C05446=1014.097,308.316,353.938,169.733,52.430,160.170
C05447=1014.104,308.600,353.902,169.740,52.424,160.169
C05448=1014.111,308.846,353.870,169.746,52.418,160.169
C05449=1014.117,309.094,353.839,169.753,52.412,160.169
C05450=1014.123,309.343,353.807,169.760,52.406,160.169
C05451=1014.128,309.590,353.774,169.766,52.401,160.169
C05452=1014.134,309.838,353.742,169.772,52.395,160.169
C05453=1014.141,310.086,353.709,169.779,52.389,160.169
C05454=1014.147,310.333,353.676,169.785,52.384,160.169
C05455=1014.153,310.581,353.644,169.792,52.379,160.169
C05456=1014.158,310.829,353.611,169.798,52.373,160.169
C05457=1014.164,311.077,353.579,169.804,52.367,160.169
C05458=1014.170,311.324,353.547,169.811,52.362,160.169
C05459=1014.176,311.572,353.514,169.817,52.356,160.169
C05460=1014.182,311.820,353.482,169.824,52.350,160.169
C05461=1014.189,312.068,353.449,169.831,52.345,160.169
C05462=1014.194,312.315,353.416,169.837,52.339,160.169
C05463=1014.200,312.563,353.384,169.843,52.333,160.169
C05464=1014.206,312.811,353.351,169.850,52.328,160.169
C05465=1014.212,313.058,353.319,169.856,52.323,160.169
C05466=1014.218,313.306,353.286,169.863,52.317,160.169
C05467=1014.224,313.554,353.254,169.869,52.311,160.169
C05468=1014.230,313.802,353.220,169.876,52.306,160.169
C05469=1014.236,314.050,353.188,169.883,52.300,160.169
C05470=1014.243,314.297,353.155,169.889,52.295,160.169
C05471=1014.249,314.545,353.122,169.896,52.290,160.169
C05472=1014.255,314.792,353.089,169.902,52.284,160.169
C05473=1014.261,315.040,353.056,169.909,52.278,160.169
C05474=1014.267,315.289,353.024,169.915,52.273,160.169
C05475=1014.273,315.536,352.991,169.922,52.268,160.169
C05476=1014.279,315.784,352.959,169.928,52.263,160.169
C05477=1014.286,316.031,352.926,169.936,52.257,160.169
C05478=1014.292,316.279,352.893,169.942,52.252,160.169
C05479=1014.297,316.527,352.860,169.949,52.246,160.169
C05480=1014.304,316.775,352.827,169.955,52.241,160.169
C05481=1014.311,317.023,352.794,169.962,52.236,160.169
C05482=1014.317,317.270,352.761,169.968,52.231,160.169
C05483=1014.323,317.518,352.728,169.975,52.225,160.169
C05484=1014.329,317.766,352.695,169.982,52.220,160.169
C05485=1014.335,318.013,352.662,169.989,52.214,160.169
C05486=1014.342,318.260,352.629,169.995,52.209,160.169
C05487=1014.348,318.509,352.596,170.002,52.203,160.169
C05488=1014.355,318.756,352.563,170.008,52.198,160.169
C05489=1014.360,319.004,352.530,170.015,52.193,160.169
C05490=1014.367,319.252,352.497,170.022,52.187,160.169
C05491=1014.374,319.499,352.463,170.029,52.182,160.169
C05492=1014.380,319.747,352.430,170.036,52.177,160.170
C05493=1014.386,319.995,352.398,170.042,52.172,160.169
C05494=1014.392,320.243,352.364,170.049,52.167,160.170
C05495=1014.399,320.490,352.331,170.056,52.162,160.170
C05496=1014.405,320.738,352.298,170.063,52.156,160.170
C05497=1014.412,320.985,352.265,170.070,52.151,160.170
C05498=1014.419,321.233,352.231,170.076,52.146,160.170
C05499=1014.425,321.481,352.198,170.083,52.141,160.170
C05500=1014.431,321.729,352.165,170.090,52.136,160.170
C05501=1014.438,321.976,352.131,170.096,52.131,160.170
C05502=1014.444,322.224,352.099,170.104,52.125,160.170
C05503=1014.452,322.472,352.065,170.110,52.120,160.170
C05504=1014.458,322.761,352.026,170.118,52.114,160.171
C05505=1014.466,323.050,351.987,170.126,52.108,160.171
C05506=1014.474,323.339,351.948,170.135,52.102,160.171
C05507=1014.481,323.628,351.909,170.143,52.096,160.171
C05508=1014.488,323.876,351.876,170.149,52.091,160.171
C05509=1014.495,324.123,351.842,170.156,52.086,160.171
C05510=1014.501,324.372,351.809,170.164,52.081,160.171
C05511=1014.507,324.619,351.775,170.170,52.076,160.172
C05512=1014.515,324.867,351.741,170.177,52.071,160.172
C05513=1014.521,325.114,351.709,170.184,52.066,160.172
C05514=1014.528,325.362,351.675,170.192,52.061,160.172
C05515=1014.535,325.609,351.641,170.198,52.056,160.172
C05516=1014.541,325.857,351.608,170.205,52.051,160.172
C05517=1014.547,326.104,351.574,170.212,52.046,160.172
C05518=1014.554,326.352,351.540,170.219,52.042,160.173
C05519=1014.560,326.600,351.505,170.226,52.037,160.173
C05520=1014.567,326.847,351.472,170.233,52.031,160.173
C05521=1014.573,327.095,351.437,170.240,52.026,160.173
C05522=1014.579,327.343,351.403,170.247,52.022,160.174
C05523=1014.586,327.590,351.369,170.254,52.017,160.174
C05524=1014.593,327.838,351.335,170.261,52.012,160.174
C05525=1014.599,328.085,351.301,170.268,52.008,160.174
C05526=1014.606,328.333,351.267,170.275,52.003,160.174
C05527=1014.612,328.580,351.232,170.283,51.998,160.175
C05528=1014.619,328.828,351.198,170.290,51.993,160.175
C05529=1014.626,329.075,351.164,170.296,51.988,160.175
C05530=1014.632,329.323,351.130,170.303,51.984,160.175
C05531=1014.638,329.571,351.096,170.310,51.979,160.175
C05532=1014.645,329.818,351.062,170.318,51.974,160.176
C05533=1014.652,330.066,351.027,170.325,51.969,160.176
C05534=1014.658,330.313,350.993,170.332,51.965,160.176
C05535=1014.665,330.561,350.959,170.339,51.960,160.176
C05536=1014.672,330.809,350.924,170.346,51.956,160.177
C05537=1014.678,331.056,350.889,170.353,51.951,160.177
C05538=1014.686,331.304,350.855,170.361,51.946,160.177
C05539=1014.691,331.551,350.821,170.368,51.942,160.178
C05540=1014.698,331.798,350.786,170.375,51.937,160.178
C05541=1014.705,332.046,350.752,170.382,51.933,160.178
C05542=1014.712,332.293,350.717,170.389,51.928,160.178
C05543=1014.719,332.541,350.683,170.397,51.923,160.178
C05544=1014.725,332.789,350.648,170.404,51.919,160.179
C05545=1014.731,333.036,350.614,170.411,51.914,160.179
C05546=1014.738,333.283,350.579,170.418,51.910,160.179
C05547=1014.745,333.531,350.543,170.425,51.905,160.180
C05548=1014.751,333.779,350.509,170.433,51.901,160.180
C05549=1014.759,334.026,350.474,170.440,51.896,160.180
C05550=1014.766,334.273,350.439,170.448,51.892,160.181
C05551=1014.772,334.521,350.405,170.455,51.888,160.181
C05552=1014.779,334.769,350.370,170.462,51.883,160.181
C05553=1014.786,335.016,350.335,170.470,51.878,160.182
C05554=1014.792,335.263,350.300,170.477,51.874,160.182
C05555=1014.799,335.511,350.265,170.484,51.870,160.182
C05556=1014.806,335.759,350.230,170.491,51.865,160.182
C05557=1014.812,336.006,350.195,170.498,51.861,160.183
C05558=1014.819,336.253,350.160,170.506,51.856,160.183
C05559=1014.826,336.501,350.125,170.513,51.852,160.184
C05560=1014.833,336.748,350.089,170.521,51.848,160.184
C05561=1014.839,336.995,350.054,170.528,51.843,160.184
C05562=1014.846,337.243,350.020,170.535,51.839,160.185
C05563=1014.853,337.491,349.985,170.543,51.834,160.185
C05564=1014.861,337.776,349.944,170.551,51.830,160.185
C05565=1014.869,338.060,349.903,170.560,51.825,160.186
C05566=1014.877,338.345,349.864,170.569,51.820,160.186
C05567=1014.885,338.630,349.823,170.578,51.815,160.187
C05568=1014.892,338.878,349.788,170.585,51.811,160.187
C05569=1014.899,339.125,349.752,170.592,51.807,160.187
C05570=1014.905,339.372,349.716,170.600,51.803,160.188
C05571=1014.912,339.619,349.681,170.608,51.798,160.188
C05572=1014.919,339.867,349.645,170.615,51.794,160.189
C05573=1014.926,340.114,349.610,170.623,51.790,160.189
C05574=1014.933,340.362,349.574,170.630,51.786,160.190
C05575=1014.940,340.609,349.539,170.638,51.781,160.190
C05576=1014.946,340.856,349.503,170.645,51.778,160.191
C05577=1014.954,341.104,349.467,170.653,51.773,160.191
C05578=1014.960,341.351,349.432,170.660,51.770,160.191
C05579=1014.967,341.598,349.396,170.668,51.765,160.192
C05580=1014.975,341.846,349.361,170.675,51.761,160.192
C05581=1014.981,342.093,349.324,170.683,51.757,160.193
C05582=1014.988,342.341,349.289,170.690,51.753,160.193
C05583=1014.996,342.588,349.253,170.699,51.749,160.194
C05584=1015.002,342.835,349.218,170.706,51.745,160.194
C05585=1015.009,343.083,349.181,170.714,51.741,160.194
C05586=1015.016,343.330,349.145,170.721,51.737,160.195
C05587=1015.023,343.577,349.110,170.729,51.733,160.195
C05588=1015.030,343.825,349.073,170.737,51.729,160.196
C05589=1015.037,344.072,349.037,170.744,51.726,160.197
C05590=1015.044,344.319,349.002,170.753,51.721,160.197
C05591=1015.052,344.567,348.966,170.760,51.717,160.197
C05592=1015.058,344.814,348.930,170.768,51.714,160.198
C05593=1015.066,345.061,348.893,170.776,51.709,160.198
C05594=1015.072,345.309,348.858,170.783,51.705,160.199
C05595=1015.080,345.556,348.822,170.791,51.702,160.199
C05596=1015.086,345.803,348.786,170.799,51.698,160.200
C05597=1015.094,346.050,348.749,170.807,51.694,160.201
C05598=1015.101,346.297,348.714,170.814,51.690,160.201
C05599=1015.108,346.545,348.677,170.822,51.686,160.201
C05600=1015.116,346.792,348.641,170.830,51.682,160.202
C05601=1015.122,347.039,348.604,170.838,51.679,160.203
C05602=1015.130,347.287,348.568,170.846,51.675,160.203
C05603=1015.137,347.534,348.532,170.854,51.671,160.204
C05604=1015.144,347.781,348.495,170.862,51.667,160.204
C05605=1015.151,348.028,348.459,170.869,51.664,160.205
C05606=1015.158,348.276,348.423,170.878,51.660,160.206
C05607=1015.165,348.523,348.385,170.886,51.656,160.206
C05608=1015.172,348.770,348.349,170.893,51.652,160.207
C05609=1015.179,349.018,348.312,170.902,51.649,160.207
C05610=1015.187,349.265,348.276,170.909,51.645,160.208
C05611=1015.193,349.511,348.239,170.917,51.641,160.208
C05612=1015.201,349.759,348.203,170.926,51.638,160.209
C05613=1015.208,350.007,348.166,170.933,51.634,160.210
C05614=1015.216,350.253,348.129,170.942,51.630,160.210
C05615=1015.222,350.500,348.093,170.950,51.627,160.211
C05616=1015.230,350.747,348.056,170.957,51.623,160.211
C05617=1015.237,350.995,348.019,170.966,51.620,160.212
C05618=1015.245,351.243,347.983,170.974,51.616,160.213
C05619=1015.252,351.490,347.945,170.981,51.612,160.213
C05620=1015.259,351.736,347.909,170.990,51.609,160.214
C05621=1015.266,351.984,347.872,170.998,51.605,160.215
C05622=1015.274,352.231,347.834,171.006,51.601,160.215
C05623=1015.281,352.478,347.798,171.014,51.598,160.216
C05624=1015.290,352.760,347.756,171.024,51.594,160.217
C05625=1015.299,353.042,347.713,171.033,51.590,160.217
C05626=1015.307,353.325,347.671,171.043,51.586,160.218
C05627=1015.315,353.607,347.629,171.052,51.582,160.219
C05628=1015.322,353.854,347.592,171.060,51.579,160.220
C05629=1015.330,354.100,347.555,171.068,51.575,160.220
C05630=1015.337,354.348,347.517,171.077,51.572,160.221
C05631=1015.344,354.595,347.480,171.084,51.568,160.222
C05632=1015.352,354.842,347.442,171.093,51.565,160.222
C05633=1015.360,355.089,347.405,171.101,51.561,160.223
C05634=1015.367,355.336,347.368,171.110,51.558,160.224
C05635=1015.374,355.584,347.331,171.118,51.555,160.224
C05636=1015.382,355.831,347.293,171.126,51.551,160.225
C05637=1015.390,356.078,347.255,171.134,51.548,160.226
C05638=1015.397,356.325,347.218,171.143,51.545,160.227
C05639=1015.405,356.572,347.180,171.151,51.542,160.227
C05640=1015.412,356.819,347.143,171.160,51.538,160.228
C05641=1015.420,357.066,347.106,171.168,51.535,160.229
C05642=1015.427,357.313,347.068,171.177,51.532,160.230
C05643=1015.434,357.560,347.031,171.185,51.529,160.230
C05644=1015.442,357.807,346.992,171.194,51.525,160.231
C05645=1015.450,358.054,346.955,171.202,51.522,160.232
C05646=1015.458,358.301,346.918,171.211,51.519,160.233
C05647=1015.465,358.548,346.880,171.219,51.516,160.233
C05648=1015.472,358.795,346.842,171.227,51.512,160.234
C05649=1015.480,359.043,346.804,171.236,51.510,160.235
C05650=1015.488,359.289,346.766,171.245,51.506,160.236
C05651=1015.495,359.536,346.728,171.253,51.503,160.237
C05652=1015.503,359.783,346.690,171.262,51.500,160.237
C05653=1015.510,360.030,346.652,171.270,51.497,160.238
C05654=1015.518,360.277,346.614,171.279,51.494,160.239
C05655=1015.525,360.524,346.576,171.287,51.491,160.240
C05656=1015.533,360.771,346.538,171.296,51.487,160.241
C05657=1015.541,361.018,346.499,171.304,51.485,160.242
C05658=1015.548,361.265,346.461,171.313,51.482,160.242
C05659=1015.556,361.512,346.424,171.322,51.478,160.243
C05660=1015.563,361.759,346.384,171.330,51.475,160.244
C05661=1015.571,362.006,346.346,171.339,51.472,160.245
C05662=1015.579,362.253,346.308,171.347,51.469,160.246
C05663=1015.586,362.500,346.270,171.356,51.466,160.247
C05664=1015.594,362.747,346.232,171.366,51.463,160.248
C05665=1015.602,362.994,346.193,171.374,51.460,160.248
C05666=1015.609,363.240,346.155,171.383,51.457,160.249
C05667=1015.617,363.488,346.116,171.391,51.455,160.250
C05668=1015.625,363.734,346.078,171.400,51.451,160.251
C05669=1015.633,363.981,346.040,171.410,51.449,160.252
C05670=1015.641,364.228,346.001,171.418,51.446,160.253
C05671=1015.649,364.475,345.963,171.427,51.443,160.254
C05672=1015.657,364.722,345.924,171.436,51.440,160.255
C05673=1015.665,364.969,345.886,171.444,51.437,160.256
C05674=1015.673,365.216,345.847,171.453,51.434,160.256
C05675=1015.680,365.463,345.809,171.463,51.431,160.257
C05676=1015.689,365.709,345.770,171.471,51.429,160.258
C05677=1015.696,365.957,345.730,171.480,51.425,160.259
C05678=1015.704,366.203,345.692,171.489,51.423,160.260
C05679=1015.712,366.450,345.654,171.499,51.420,160.261
C05680=1015.720,366.697,345.614,171.507,51.417,160.262
C05681=1015.728,366.944,345.576,171.516,51.414,160.263
C05682=1015.736,367.191,345.537,171.526,51.412,160.264
C05683=1015.744,367.437,345.498,171.534,51.409,160.265
C05684=1015.753,367.727,345.452,171.545,51.406,160.266
C05685=1015.763,368.017,345.406,171.556,51.403,160.267
C05686=1015.772,368.307,345.361,171.566,51.400,160.268
C05687=1015.781,368.596,345.315,171.577,51.396,160.270
C05688=1015.789,368.843,345.275,171.586,51.394,160.271
C05689=1015.797,369.090,345.236,171.595,51.391,160.272
C05690=1015.806,369.336,345.196,171.605,51.388,160.273
C05691=1015.813,369.584,345.157,171.613,51.386,160.274
C05692=1015.821,369.831,345.118,171.623,51.383,160.275
C05693=1015.829,370.077,345.078,171.632,51.380,160.276
C05694=1015.837,370.323,345.039,171.642,51.378,160.277
C05695=1015.845,370.570,345.000,171.651,51.376,160.278
C05696=1015.853,370.817,344.960,171.660,51.373,160.279
C05697=1015.861,371.064,344.921,171.669,51.371,160.280
C05698=1015.869,371.311,344.881,171.678,51.368,160.281
C05699=1015.878,371.558,344.842,171.688,51.366,160.282
C05700=1015.886,371.804,344.803,171.698,51.363,160.283
C05701=1015.894,372.051,344.763,171.707,51.360,160.284
C05702=1015.902,372.298,344.723,171.715,51.358,160.285
C05703=1015.911,372.544,344.683,171.725,51.356,160.287
C05704=1015.919,372.791,344.643,171.735,51.353,160.288
C05705=1015.927,373.037,344.604,171.744,51.351,160.289
C05706=1015.935,373.284,344.564,171.754,51.348,160.290
C05707=1015.943,373.531,344.525,171.763,51.346,160.291
C05708=1015.952,373.778,344.485,171.773,51.343,160.292
C05709=1015.960,374.024,344.444,171.782,51.341,160.293
C05710=1015.969,374.271,344.405,171.792,51.339,160.294
C05711=1015.977,374.518,344.365,171.801,51.336,160.295
C05712=1015.985,374.764,344.325,171.811,51.334,160.297
C05713=1015.994,375.011,344.285,171.821,51.332,160.298
C05714=1016.002,375.258,344.246,171.830,51.329,160.299
C05715=1016.011,375.504,344.205,171.840,51.327,160.300
C05716=1016.019,375.751,344.166,171.850,51.325,160.302
C05717=1016.027,375.998,344.125,171.859,51.322,160.303
C05718=1016.036,376.244,344.085,171.868,51.320,160.304
C05719=1016.044,376.491,344.045,171.878,51.318,160.305
C05720=1016.052,376.737,344.004,171.888,51.316,160.306
C05721=1016.060,376.984,343.963,171.898,51.314,160.307
C05722=1016.069,377.230,343.923,171.907,51.311,160.308
C05723=1016.077,377.476,343.882,171.917,51.309,160.310
C05724=1016.085,377.724,343.842,171.927,51.307,160.311
C05725=1016.093,377.970,343.801,171.937,51.304,160.312
C05726=1016.102,378.216,343.761,171.947,51.302,160.314
C05727=1016.111,378.463,343.720,171.957,51.300,160.315
C05728=1016.119,378.709,343.680,171.967,51.298,160.316
C05729=1016.128,378.956,343.639,171.977,51.296,160.317
C05730=1016.136,379.202,343.599,171.986,51.294,160.319
C05731=1016.145,379.449,343.558,171.997,51.292,160.320
C05732=1016.153,379.696,343.517,172.006,51.290,160.321
C05733=1016.163,379.942,343.476,172.016,51.288,160.323
C05734=1016.171,380.188,343.435,172.026,51.286,160.324
C05735=1016.179,380.435,343.394,172.036,51.284,160.325
C05736=1016.187,380.681,343.354,172.047,51.282,160.327
C05737=1016.197,380.928,343.313,172.057,51.280,160.328
C05738=1016.206,381.174,343.272,172.067,51.278,160.329
C05739=1016.214,381.421,343.231,172.076,51.276,160.330
C05740=1016.222,381.668,343.190,172.087,51.274,160.332
C05741=1016.231,381.913,343.149,172.097,51.272,160.333
C05742=1016.240,382.160,343.108,172.108,51.270,160.335
C05743=1016.249,382.407,343.067,172.117,51.268,160.336
C05744=1016.260,382.719,343.015,172.130,51.265,160.338
C05745=1016.271,383.031,342.963,172.143,51.263,160.339
C05746=1016.282,383.343,342.910,172.156,51.261,160.341
C05747=1016.294,383.656,342.859,172.169,51.258,160.343
C05748=1016.303,383.903,342.817,172.179,51.256,160.344
C05749=1016.311,384.148,342.776,172.190,51.254,160.346
C05750=1016.321,384.395,342.735,172.201,51.253,160.347
C05751=1016.330,384.641,342.693,172.210,51.251,160.348
C05752=1016.338,384.888,342.652,172.222,51.249,160.350
C05753=1016.347,385.134,342.610,172.232,51.247,160.351
C05754=1016.356,385.381,342.568,172.242,51.246,160.353
C05755=1016.365,385.627,342.527,172.253,51.243,160.354
C05756=1016.374,385.873,342.485,172.263,51.242,160.356
C05757=1016.383,386.120,342.443,172.273,51.240,160.357
C05758=1016.392,386.366,342.401,172.284,51.238,160.359
C05759=1016.401,386.612,342.360,172.295,51.237,160.360
C05760=1016.409,386.858,342.318,172.305,51.235,160.362
C05761=1016.419,387.105,342.276,172.316,51.234,160.363
C05762=1016.428,387.351,342.235,172.326,51.232,160.365
C05763=1016.437,387.598,342.193,172.337,51.230,160.366
C05764=1016.446,387.844,342.150,172.348,51.229,160.368
C05765=1016.455,388.090,342.109,172.359,51.227,160.369
C05766=1016.464,388.336,342.066,172.369,51.226,160.371
C05767=1016.473,388.582,342.025,172.380,51.224,160.372
C05768=1016.482,388.828,341.983,172.391,51.222,160.374
C05769=1016.490,389.074,341.940,172.401,51.221,160.375
C05770=1016.499,389.321,341.898,172.413,51.220,160.377
C05771=1016.509,389.567,341.855,172.423,51.218,160.378
C05772=1016.519,389.813,341.813,172.434,51.216,160.380
C05773=1016.527,390.059,341.771,172.446,51.215,160.382
C05774=1016.537,390.305,341.729,172.456,51.213,160.383
C05775=1016.547,390.552,341.686,172.467,51.212,160.385
C05776=1016.555,390.798,341.644,172.478,51.210,160.386
C05777=1016.564,391.044,341.601,172.489,51.209,160.388
C05778=1016.574,391.290,341.558,172.499,51.208,160.390
C05779=1016.583,391.536,341.516,172.511,51.206,160.391
C05780=1016.592,391.783,341.474,172.522,51.204,160.393
C05781=1016.602,392.029,341.431,172.533,51.203,160.395
C05782=1016.610,392.275,341.388,172.544,51.202,160.396
C05783=1016.620,392.522,341.346,172.555,51.200,160.398
C05784=1016.630,392.767,341.302,172.566,51.199,160.400
C05785=1016.639,393.012,341.260,172.578,51.198,160.401
C05786=1016.648,393.259,341.217,172.589,51.197,160.403
C05787=1016.657,393.505,341.174,172.599,51.195,160.405
C05788=1016.667,393.751,341.131,172.611,51.194,160.406
C05789=1016.676,393.997,341.088,172.623,51.192,160.408
C05790=1016.686,394.243,341.045,172.633,51.192,160.410
C05791=1016.696,394.490,341.002,172.645,51.190,160.412
C05792=1016.704,394.736,340.959,172.656,51.189,160.413
C05793=1016.714,394.982,340.916,172.668,51.188,160.415
C05794=1016.724,395.227,340.873,172.680,51.186,160.417
C05795=1016.733,395.473,340.829,172.690,51.185,160.419
C05796=1016.743,395.720,340.786,172.702,51.184,160.420
C05797=1016.752,395.965,340.743,172.713,51.183,160.422
C05798=1016.761,396.212,340.700,172.725,51.182,160.424
C05799=1016.772,396.458,340.656,172.737,51.181,160.426
C05800=1016.782,396.703,340.613,172.749,51.179,160.428
C05801=1016.790,396.949,340.570,172.760,51.178,160.429
C05802=1016.800,397.195,340.526,172.771,51.178,160.431
C05803=1016.810,397.441,340.482,172.783,51.176,160.433
C05804=1016.824,397.787,340.421,172.799,51.175,160.436
C05805=1016.837,398.133,340.359,172.816,51.174,160.438
C05806=1016.851,398.479,340.298,172.832,51.172,160.441
C05807=1016.865,398.826,340.236,172.849,51.170,160.443
C05808=1016.874,399.071,340.193,172.861,51.170,160.445
C05809=1016.884,399.318,340.149,172.873,51.169,160.447
C05810=1016.894,399.563,340.105,172.884,51.168,160.449
C05811=1016.904,399.809,340.060,172.896,51.167,160.451
C05812=1016.914,400.055,340.017,172.909,51.166,160.453
C05813=1016.923,400.301,339.973,172.921,51.164,160.455
C05814=1016.934,400.547,339.927,172.933,51.164,160.457
C05815=1016.943,400.793,339.883,172.945,51.163,160.459
C05816=1016.953,401.038,339.839,172.957,51.162,160.461
C05817=1016.963,401.285,339.795,172.969,51.161,160.463
C05818=1016.973,401.530,339.750,172.981,51.161,160.465
C05819=1016.983,401.776,339.707,172.993,51.160,160.467
C05820=1016.992,402.021,339.662,173.005,51.159,160.469
C05821=1017.002,402.268,339.618,173.018,51.158,160.471
C05822=1017.012,402.514,339.573,173.030,51.157,160.473
C05823=1017.023,402.759,339.528,173.042,51.156,160.475
C05824=1017.032,403.004,339.483,173.054,51.156,160.477
C05825=1017.042,403.251,339.439,173.066,51.156,160.479
C05826=1017.053,403.497,339.395,173.079,51.154,160.481
C05827=1017.062,403.742,339.350,173.091,51.154,160.483
C05828=1017.072,403.988,339.305,173.103,51.153,160.485
C05829=1017.083,404.233,339.261,173.117,51.152,160.487
C05830=1017.093,404.479,339.216,173.129,51.152,160.489
C05831=1017.103,404.724,339.171,173.141,51.151,160.491
C05832=1017.113,404.971,339.126,173.154,51.150,160.493
C05833=1017.123,405.216,339.081,173.166,51.149,160.495
C05834=1017.134,405.461,339.036,173.178,51.149,160.498
C05835=1017.144,405.707,338.991,173.192,51.149,160.500
C05836=1017.155,405.953,338.946,173.204,51.148,160.502
C05837=1017.165,406.198,338.901,173.217,51.147,160.504
C05838=1017.175,406.444,338.855,173.229,51.147,160.506
C05839=1017.186,406.690,338.811,173.242,51.146,160.508
C05840=1016.824,404.675,338.837,173.123,51.219,160.507
C05841=1016.814,404.429,338.882,173.110,51.220,160.505
C05842=1016.804,404.183,338.927,173.097,51.220,160.502
C05843=1016.793,403.938,338.971,173.085,51.221,160.500
C05844=1016.784,403.692,339.016,173.072,51.222,160.498
C05845=1016.773,403.446,339.061,173.060,51.223,160.496
C05846=1016.763,403.201,339.106,173.048,51.223,160.494
C05847=1016.753,402.955,339.150,173.035,51.224,160.492
C05848=1016.744,402.709,339.195,173.023,51.225,160.490
C05849=1016.733,402.463,339.239,173.011,51.226,160.488
C05850=1016.723,402.217,339.283,172.998,51.227,160.486
C05851=1016.714,401.972,339.328,172.986,51.228,160.484
C05852=1016.704,401.726,339.373,172.974,51.229,160.482
C05853=1016.694,401.480,339.416,172.962,51.229,160.480
C05854=1016.684,401.235,339.461,172.950,51.230,160.478
C05855=1016.675,400.989,339.505,172.937,51.231,160.476
C05856=1016.664,400.744,339.550,172.925,51.232,160.474
C05857=1016.654,400.497,339.594,172.914,51.234,160.473
C05858=1016.645,400.251,339.638,172.902,51.234,160.471
C05859=1016.634,400.005,339.682,172.890,51.235,160.469
C05860=1016.625,399.759,339.727,172.878,51.236,160.467
C05861=1016.615,399.513,339.771,172.866,51.237,160.465
C05862=1016.605,399.267,339.814,172.853,51.238,160.463
C05863=1016.596,399.021,339.858,172.842,51.240,160.461
C05864=1016.586,398.776,339.901,172.830,51.240,160.459
C05865=1016.574,398.464,339.958,172.816,51.242,160.457
C05866=1016.561,398.152,340.013,172.800,51.243,160.454
C05867=1016.550,397.839,340.068,172.785,51.245,160.452
C05868=1016.537,397.528,340.124,172.770,51.246,160.450
C05869=1016.527,397.282,340.168,172.758,51.248,160.448
C05870=1016.518,397.036,340.211,172.747,51.249,160.446
C05871=1016.508,396.790,340.254,172.736,51.249,160.444
C05872=1016.498,396.544,340.298,172.724,51.251,160.442
C05873=1016.489,396.297,340.341,172.712,51.252,160.441
C05874=1016.479,396.052,340.384,172.701,51.253,160.439
C05875=1016.470,395.805,340.428,172.689,51.255,160.437
C05876=1016.460,395.560,340.471,172.678,51.256,160.435
C05877=1016.451,395.314,340.513,172.666,51.257,160.434
C05878=1016.441,395.068,340.558,172.654,51.259,160.432
C05879=1016.431,394.821,340.600,172.643,51.260,160.430
C05880=1016.422,394.576,340.644,172.631,51.261,160.428
C05881=1016.412,394.330,340.686,172.621,51.262,160.427
C05882=1016.403,394.084,340.729,172.609,51.264,160.425
C05883=1016.394,393.837,340.772,172.598,51.266,160.423
C05884=1016.384,393.592,340.815,172.586,51.267,160.422
C05885=1016.375,393.345,340.859,172.575,51.268,160.420
C05886=1016.366,393.100,340.901,172.564,51.269,160.418
C05887=1016.356,392.853,340.944,172.553,51.271,160.417
C05888=1016.347,392.607,340.987,172.541,51.272,160.415
C05889=1016.338,392.361,341.030,172.530,51.274,160.413
C05890=1016.328,392.115,341.072,172.519,51.275,160.411
C05891=1016.320,391.869,341.115,172.508,51.277,160.410
C05892=1016.310,391.622,341.158,172.497,51.279,160.408
C05893=1016.301,391.377,341.200,172.486,51.279,160.406
C05894=1016.292,391.130,341.242,172.475,51.281,160.405
C05895=1016.282,390.884,341.285,172.463,51.283,160.403
C05896=1016.273,390.638,341.327,172.453,51.284,160.402
C05897=1016.263,390.392,341.370,172.442,51.286,160.400
C05898=1016.254,390.145,341.412,172.430,51.287,160.398
C05899=1016.245,389.899,341.455,172.420,51.289,160.397
C05900=1016.237,389.653,341.497,172.409,51.291,160.395
C05901=1016.227,389.407,341.539,172.398,51.293,160.394
C05902=1016.218,389.161,341.581,172.387,51.294,160.392
C05903=1016.209,388.914,341.624,172.376,51.296,160.391
C05904=1016.200,388.668,341.665,172.366,51.297,160.389
C05905=1016.190,388.422,341.708,172.355,51.299,160.388
C05906=1016.181,388.176,341.749,172.344,51.301,160.386
C05907=1016.173,387.930,341.792,172.333,51.303,160.385
C05908=1016.164,387.683,341.834,172.323,51.304,160.383
C05909=1016.155,387.437,341.876,172.312,51.306,160.382
C05910=1016.146,387.191,341.918,172.302,51.308,160.380
C05911=1016.137,386.944,341.959,172.290,51.309,160.379
C05912=1016.128,386.698,342.001,172.280,51.311,160.377
C05913=1016.119,386.452,342.043,172.269,51.313,160.375
C05914=1016.110,386.206,342.085,172.259,51.314,160.374
C05915=1016.101,385.959,342.127,172.248,51.317,160.373
C05916=1016.092,385.713,342.169,172.238,51.319,160.371
C05917=1016.083,385.467,342.210,172.227,51.320,160.370
C05918=1016.075,385.220,342.251,172.216,51.322,160.368
C05919=1016.065,384.974,342.292,172.207,51.324,160.367
C05920=1016.057,384.728,342.334,172.195,51.326,160.365
C05921=1016.048,384.482,342.376,172.185,51.328,160.364
C05922=1016.039,384.235,342.417,172.174,51.330,160.363
C05923=1016.030,383.988,342.458,172.164,51.332,160.361
C05924=1016.020,383.742,342.499,172.154,51.334,160.360
C05925=1016.010,383.427,342.552,172.141,51.336,160.358
C05926=1015.998,383.113,342.605,172.128,51.338,160.356
C05927=1015.987,382.798,342.657,172.114,51.341,160.354
C05928=1015.975,382.483,342.709,172.101,51.344,160.353
C05929=1015.967,382.236,342.750,172.091,51.346,160.351
C05930=1015.958,381.991,342.792,172.081,51.348,160.350
C05931=1015.950,381.744,342.833,172.070,51.350,160.349
C05932=1015.940,381.497,342.873,172.061,51.352,160.347
C05933=1015.932,381.251,342.914,172.051,51.354,160.346
C05934=1015.923,381.004,342.955,172.040,51.357,160.345
C05935=1015.915,380.758,342.995,172.030,51.359,160.344
C05936=1015.906,380.511,343.036,172.020,51.360,160.342
C05937=1015.898,380.266,343.078,172.010,51.362,160.341
C05938=1015.889,380.019,343.119,171.999,51.365,160.340
C05939=1015.880,379.772,343.159,171.990,51.367,160.338
C05940=1015.872,379.526,343.200,171.980,51.369,160.337
C05941=1015.864,379.279,343.240,171.970,51.371,160.336
C05942=1015.855,379.032,343.281,171.960,51.373,160.335
C05943=1015.846,378.787,343.321,171.950,51.376,160.333
C05944=1015.838,378.540,343.362,171.940,51.378,160.332
C05945=1015.830,378.293,343.403,171.930,51.380,160.331
C05946=1015.820,378.047,343.443,171.920,51.382,160.329
C05947=1015.812,377.800,343.484,171.910,51.384,160.328
C05948=1015.805,377.553,343.524,171.901,51.387,160.327
C05949=1015.796,377.306,343.565,171.891,51.389,160.326
C05950=1015.787,377.060,343.605,171.881,51.391,160.325
C05951=1015.779,376.814,343.646,171.871,51.394,160.323
C05952=1015.771,376.567,343.686,171.862,51.396,160.322
C05953=1015.763,376.320,343.727,171.852,51.398,160.321
C05954=1015.754,376.074,343.767,171.841,51.401,160.320
C05955=1015.746,375.827,343.807,171.832,51.403,160.318
C05956=1015.738,375.581,343.847,171.822,51.406,160.317
C05957=1015.729,375.334,343.888,171.813,51.408,160.316
C05958=1015.721,375.088,343.928,171.803,51.411,160.315
C05959=1015.713,374.841,343.967,171.793,51.413,160.314
C05960=1015.705,374.595,344.007,171.784,51.416,160.313
C05961=1015.696,374.348,344.047,171.774,51.418,160.312
C05962=1015.687,374.101,344.086,171.765,51.420,160.311
C05963=1015.679,373.854,344.126,171.755,51.423,160.309
C05964=1015.671,373.608,344.166,171.746,51.425,160.308
C05965=1015.662,373.361,344.206,171.736,51.428,160.307
C05966=1015.655,373.114,344.246,171.726,51.430,160.306
C05967=1015.646,372.868,344.285,171.717,51.433,160.305
C05968=1015.638,372.621,344.325,171.708,51.436,160.304
C05969=1015.630,372.374,344.364,171.698,51.438,160.303
C05970=1015.621,372.128,344.404,171.688,51.440,160.302
C05971=1015.614,371.881,344.444,171.679,51.443,160.301
C05972=1015.605,371.634,344.483,171.670,51.446,160.299
C05973=1015.598,371.387,344.523,171.661,51.448,160.299
C05974=1015.589,371.141,344.562,171.652,51.451,160.298
C05975=1015.581,370.894,344.601,171.642,51.454,160.296
C05976=1015.573,370.647,344.641,171.633,51.456,160.295
C05977=1015.564,370.401,344.681,171.623,51.459,160.294
C05978=1015.557,370.154,344.721,171.614,51.461,160.293
C05979=1015.549,369.906,344.759,171.604,51.464,160.292
C05980=1015.541,369.661,344.798,171.595,51.467,160.291
C05981=1015.533,369.414,344.838,171.587,51.469,160.290
C05982=1015.525,369.166,344.877,171.577,51.472,160.289
C05983=1015.516,368.920,344.916,171.568,51.475,160.288
C05984=1015.509,368.673,344.956,171.559,51.478,160.287
C05985=1015.500,368.381,345.002,171.549,51.481,160.286
C05986=1015.491,368.089,345.048,171.537,51.485,160.285
C05987=1015.481,367.797,345.094,171.527,51.488,160.284
C05988=1015.471,367.505,345.141,171.515,51.491,160.282
C05989=1015.464,367.258,345.180,171.507,51.494,160.281
C05990=1015.456,367.011,345.219,171.498,51.496,160.280
C05991=1015.448,366.765,345.257,171.489,51.500,160.280
C05992=1015.440,366.518,345.296,171.479,51.502,160.279
C05993=1015.431,366.271,345.335,171.470,51.505,160.278
C05994=1015.424,366.024,345.374,171.462,51.508,160.277
C05995=1015.416,365.777,345.412,171.452,51.511,160.276
C05996=1015.408,365.530,345.451,171.443,51.514,160.275
C05997=1015.400,365.284,345.489,171.434,51.517,160.274
C05998=1015.392,365.036,345.528,171.425,51.520,160.273
C05999=1015.384,364.790,345.566,171.417,51.523,160.272
C06000=1015.376,364.543,345.604,171.408,51.526,160.271
C06001=1015.369,364.296,345.643,171.398,51.529,160.270
C06002=1015.361,364.049,345.682,171.390,51.532,160.269
C06003=1015.353,363.801,345.721,171.381,51.535,160.269
C06004=1015.346,363.555,345.759,171.372,51.538,160.268
C06005=1015.338,363.308,345.797,171.363,51.541,160.267
C06006=1015.330,363.061,345.836,171.355,51.544,160.266
C06007=1015.322,362.815,345.874,171.346,51.547,160.265
C06008=1015.314,362.567,345.912,171.337,51.550,160.264
C06009=1015.307,362.321,345.951,171.329,51.553,160.263
C06010=1015.299,362.073,345.989,171.320,51.557,160.263
C06011=1015.291,361.826,346.027,171.310,51.560,160.262
C06012=1015.284,361.580,346.065,171.302,51.563,160.261
C06013=1015.275,361.333,346.104,171.293,51.566,160.260
C06014=1015.268,361.086,346.141,171.284,51.569,160.259
C06015=1015.261,360.839,346.179,171.276,51.572,160.258
C06016=1015.253,360.591,346.217,171.267,51.576,160.258
C06017=1015.245,360.345,346.256,171.258,51.579,160.257
C06018=1015.238,360.098,346.294,171.250,51.581,160.256
C06019=1015.230,359.851,346.331,171.241,51.585,160.255
C06020=1015.223,359.604,346.371,171.233,51.588,160.254
C06021=1015.216,359.356,346.408,171.224,51.591,160.253
C06022=1015.208,359.110,346.446,171.215,51.594,160.252
C06023=1015.201,358.863,346.484,171.207,51.598,160.252
C06024=1015.194,358.616,346.521,171.198,51.601,160.251
C06025=1015.185,358.369,346.559,171.190,51.604,160.250
C06026=1015.178,358.122,346.597,171.181,51.608,160.250
C06027=1015.170,357.874,346.634,171.172,51.611,160.249
C06028=1015.163,357.627,346.672,171.164,51.614,160.248
C06029=1015.155,357.381,346.710,171.156,51.618,160.247
C06030=1015.148,357.134,346.747,171.148,51.621,160.247
C06031=1015.140,356.886,346.785,171.139,51.625,160.246
C06032=1015.133,356.639,346.823,171.131,51.627,160.245
C06033=1015.125,356.392,346.860,171.122,51.632,160.244
C06034=1015.117,356.145,346.897,171.113,51.635,160.244
C06035=1015.110,355.898,346.935,171.106,51.639,160.243
C06036=1015.103,355.651,346.972,171.097,51.642,160.242
C06037=1015.095,355.404,347.009,171.089,51.645,160.241
C06038=1015.088,355.157,347.047,171.080,51.649,160.241
C06039=1015.080,354.910,347.084,171.072,51.652,160.240
C06040=1015.073,354.663,347.122,171.064,51.656,160.239
C06041=1015.065,354.415,347.158,171.056,51.659,160.239
C06042=1015.058,354.168,347.195,171.047,51.663,160.238
C06043=1015.051,353.921,347.233,171.039,51.666,160.237
C06044=1015.044,353.674,347.270,171.031,51.670,160.237
C06045=1015.035,353.390,347.313,171.021,51.674,160.236
C06046=1015.027,353.105,347.356,171.012,51.678,160.235
C06047=1015.018,352.821,347.398,171.002,51.682,160.234
C06048=1015.010,352.536,347.440,170.993,51.686,160.234
C06049=1015.003,352.289,347.478,170.985,51.690,160.233
C06050=1014.995,352.042,347.514,170.976,51.693,160.232
C06051=1014.988,351.795,347.551,170.969,51.697,160.232
C06052=1014.981,351.548,347.587,170.960,51.701,160.231
C06053=1014.973,351.301,347.625,170.953,51.705,160.231
C06054=1014.966,351.053,347.661,170.944,51.708,160.230
C06055=1014.958,350.806,347.698,170.936,51.712,160.229
C06056=1014.951,350.559,347.735,170.927,51.716,160.229
C06057=1014.944,350.312,347.772,170.920,51.719,160.228
C06058=1014.937,350.065,347.808,170.911,51.723,160.228
C06059=1014.930,349.817,347.845,170.904,51.727,160.227
C06060=1014.922,349.570,347.881,170.895,51.731,160.226
C06061=1014.915,349.323,347.918,170.888,51.735,160.226
C06062=1014.908,349.075,347.955,170.880,51.738,160.225
C06063=1014.901,348.829,347.991,170.871,51.742,160.225
C06064=1014.894,348.581,348.028,170.864,51.746,160.224
C06065=1014.886,348.334,348.065,170.855,51.750,160.223
C06066=1014.880,348.087,348.101,170.848,51.754,160.223
C06067=1014.872,347.840,348.137,170.840,51.757,160.222
C06068=1014.865,347.592,348.174,170.832,51.761,160.222
C06069=1014.858,347.345,348.210,170.824,51.765,160.221
C06070=1014.851,347.097,348.247,170.815,51.769,160.221
C06071=1014.844,346.851,348.283,170.808,51.772,160.220
C06072=1014.837,346.603,348.319,170.801,51.777,160.220
C06073=1014.830,346.356,348.355,170.792,51.781,160.219
C06074=1014.823,346.109,348.391,170.785,51.784,160.219
C06075=1014.816,345.862,348.427,170.776,51.788,160.218
C06076=1014.809,345.614,348.464,170.769,51.793,160.218
C06077=1014.802,345.367,348.499,170.761,51.796,160.217
C06078=1014.794,345.119,348.535,170.753,51.800,160.216
C06079=1014.788,344.872,348.572,170.746,51.805,160.216
C06080=1014.780,344.625,348.608,170.737,51.809,160.216
C06081=1014.773,344.377,348.643,170.729,51.812,160.215
C06082=1014.766,344.130,348.679,170.722,51.817,160.215
C06083=1014.759,343.883,348.716,170.714,51.821,160.214
C06084=1014.753,343.636,348.751,170.707,51.825,160.214
C06085=1014.745,343.388,348.787,170.699,51.829,160.213
C06086=1014.738,343.141,348.822,170.691,51.833,160.213
C06087=1014.732,342.894,348.859,170.683,51.837,160.212
C06088=1014.724,342.646,348.895,170.676,51.841,160.212
C06089=1014.717,342.399,348.930,170.668,51.845,160.211
C06090=1014.710,342.152,348.966,170.660,51.849,160.211
C06091=1014.704,341.904,349.002,170.652,51.853,160.210
C06092=1014.697,341.656,349.037,170.645,51.858,160.210
C06093=1014.690,341.410,349.073,170.638,51.862,160.210
C06094=1014.682,341.162,349.109,170.629,51.866,160.209
C06095=1014.675,340.915,349.144,170.622,51.870,160.209
C06096=1014.669,340.667,349.180,170.615,51.875,160.208
C06097=1014.663,340.420,349.215,170.607,51.878,160.208
C06098=1014.656,340.172,349.250,170.599,51.883,160.207
C06099=1014.648,339.925,349.287,170.592,51.887,160.207
C06100=1014.641,339.678,349.322,170.585,51.892,160.207
C06101=1014.635,339.430,349.357,170.576,51.896,160.206
C06102=1014.629,339.183,349.393,170.569,51.900,160.206
C06103=1014.621,338.936,349.429,170.562,51.904,160.205
C06104=1014.615,338.689,349.464,170.554,51.909,160.205
C06105=1014.607,338.401,349.504,170.545,51.914,160.205
C06106=1014.598,338.114,349.546,170.536,51.919,160.204
C06107=1014.590,337.826,349.586,170.528,51.924,160.204
C06108=1014.582,337.540,349.627,170.519,51.929,160.203
C06109=1014.576,337.292,349.662,170.511,51.934,160.203
C06110=1014.569,337.044,349.697,170.504,51.938,160.203
C06111=1014.562,336.797,349.732,170.497,51.942,160.202
C06112=1014.556,336.550,349.767,170.490,51.947,160.202
C06113=1014.549,336.302,349.802,170.482,51.951,160.202
C06114=1014.542,336.055,349.837,170.474,51.956,160.201
C06115=1014.535,335.808,349.872,170.467,51.960,160.201
C06116=1014.529,335.560,349.907,170.459,51.965,160.200
C06117=1014.521,335.312,349.941,170.452,51.969,160.200
C06118=1014.515,335.065,349.976,170.445,51.974,160.200
C06119=1014.508,334.818,350.012,170.437,51.978,160.200
C06120=1014.501,334.570,350.046,170.430,51.983,160.199
C06121=1014.495,334.322,350.081,170.423,51.987,160.199
C06122=1014.488,334.075,350.116,170.416,51.992,160.199
C06123=1014.481,333.827,350.151,170.408,51.997,160.198
C06124=1014.475,333.580,350.185,170.401,52.001,160.198
C06125=1014.469,333.332,350.220,170.394,52.005,160.198
C06126=1014.462,333.085,350.255,170.387,52.010,160.198
C06127=1014.455,332.838,350.290,170.379,52.015,160.197
C06128=1014.449,332.590,350.325,170.372,52.019,160.197
C06129=1014.442,332.342,350.360,170.365,52.024,160.197
C06130=1014.435,332.095,350.393,170.358,52.029,160.196
C06131=1014.429,331.847,350.428,170.350,52.034,160.196
C06132=1014.422,331.600,350.463,170.343,52.038,160.196
C06133=1014.415,331.352,350.497,170.336,52.043,160.195
C06134=1014.408,331.104,350.531,170.329,52.047,160.195
C06135=1014.402,330.858,350.566,170.321,52.052,160.195
C06136=1014.395,330.610,350.600,170.314,52.057,160.195
C06137=1014.389,330.362,350.634,170.307,52.062,160.195
C06138=1014.382,330.114,350.668,170.299,52.067,160.194
C06139=1014.375,329.868,350.703,170.293,52.072,160.194
C06140=1014.369,329.620,350.737,170.285,52.076,160.194
C06141=1014.362,329.372,350.771,170.279,52.081,160.194
C06142=1014.356,329.125,350.805,170.271,52.086,160.194
C06143=1014.349,328.877,350.839,170.264,52.091,160.193
C06144=1014.343,328.629,350.874,170.257,52.096,160.193
C06145=1014.336,328.382,350.907,170.250,52.101,160.193
C06146=1014.330,328.134,350.942,170.242,52.105,160.193
C06147=1014.324,327.887,350.976,170.236,52.110,160.192
C06148=1014.317,327.639,351.009,170.229,52.115,160.192
C06149=1014.310,327.391,351.044,170.222,52.120,160.192
C06150=1014.304,327.144,351.078,170.215,52.125,160.192
C06151=1014.297,326.896,351.112,170.207,52.130,160.192
C06152=1014.291,326.649,351.146,170.200,52.135,160.191
C06153=1014.285,326.401,351.180,170.194,52.140,160.191
C06154=1014.278,326.154,351.214,170.187,52.144,160.191
C06155=1014.272,325.906,351.248,170.179,52.150,160.191
C06156=1014.265,325.659,351.282,170.172,52.155,160.191
C06157=1014.259,325.410,351.315,170.165,52.160,160.191
C06158=1014.252,325.163,351.349,170.159,52.165,160.190
C06159=1014.245,324.915,351.383,170.151,52.170,160.190
C06160=1014.239,324.668,351.415,170.144,52.175,160.190
C06161=1014.232,324.420,351.449,170.138,52.180,160.190
C06162=1014.226,324.172,351.482,170.130,52.186,160.190
C06163=1014.219,323.925,351.516,170.124,52.191,160.190
C06164=1014.213,323.677,351.549,170.117,52.196,160.190
C06165=1014.205,323.385,351.589,170.108,52.202,160.189
C06166=1014.197,323.094,351.627,170.100,52.208,160.189
C06167=1014.190,322.803,351.667,170.093,52.214,160.189
C06168=1014.182,322.511,351.707,170.084,52.220,160.189
C06169=1014.175,322.264,351.740,170.078,52.225,160.189
C06170=1014.168,322.016,351.773,170.071,52.230,160.189
C06171=1014.162,321.769,351.806,170.063,52.236,160.189
C06172=1014.156,321.521,351.839,170.057,52.241,160.189
C06173=1014.149,321.272,351.873,170.050,52.246,160.189
C06174=1014.143,321.025,351.906,170.042,52.252,160.188
C06175=1014.137,320.778,351.939,170.036,52.257,160.188
C06176=1014.130,320.530,351.971,170.029,52.262,160.188
C06177=1014.123,320.282,352.005,170.023,52.267,160.188
C06178=1014.118,320.035,352.039,170.016,52.272,160.188
C06179=1014.111,319.787,352.071,170.009,52.278,160.188
C06180=1014.105,319.539,352.104,170.002,52.283,160.188
C06181=1014.098,319.291,352.137,169.996,52.289,160.188
C06182=1014.092,319.044,352.170,169.989,52.294,160.188
C06183=1014.086,318.796,352.204,169.981,52.299,160.188
C06184=1014.080,318.549,352.237,169.975,52.305,160.188
C06185=1014.073,318.301,352.270,169.968,52.310,160.188
C06186=1014.066,318.053,352.303,169.962,52.316,160.188
C06187=1014.060,317.805,352.335,169.954,52.321,160.188
C06188=1014.055,317.557,352.369,169.948,52.327,160.188
C06189=1014.048,317.310,352.401,169.941,52.332,160.188
C06190=1014.042,317.062,352.434,169.935,52.337,160.188
C06191=1014.036,316.815,352.467,169.928,52.342,160.188
C06192=1014.029,316.567,352.500,169.921,52.349,160.188
C06193=1014.024,316.319,352.533,169.915,52.354,160.188
C06194=1014.018,316.071,352.566,169.908,52.359,160.188
C06195=1014.011,315.824,352.598,169.902,52.365,160.188
C06196=1014.004,315.576,352.632,169.894,52.370,160.187
C06197=1013.998,315.327,352.664,169.888,52.376,160.187
C06198=1013.992,315.080,352.696,169.882,52.382,160.188
C06199=1013.987,314.832,352.730,169.875,52.387,160.187
C06200=1013.980,314.584,352.762,169.869,52.392,160.188
C06201=1013.975,314.337,352.795,169.861,52.398,160.188
C06202=1013.968,314.090,352.828,169.855,52.403,160.187
C06203=1013.962,313.842,352.860,169.848,52.409,160.187
C06204=1013.957,313.594,352.893,169.842,52.415,160.188
C06205=1013.950,313.346,352.926,169.836,52.420,160.188
C06206=1013.944,313.098,352.958,169.829,52.426,160.188
C06207=1013.938,312.850,352.990,169.822,52.431,160.187
C06208=1013.932,312.603,353.023,169.815,52.437,160.188
C06209=1013.926,312.355,353.056,169.809,52.443,160.188
C06210=1013.920,312.107,353.089,169.803,52.449,160.188
C06211=1013.915,311.860,353.121,169.797,52.454,160.188
C06212=1013.908,311.612,353.154,169.789,52.460,160.188
C06213=1013.902,311.364,353.186,169.783,52.465,160.188
C06214=1013.896,311.116,353.218,169.776,52.471,160.188
C06215=1013.890,310.868,353.250,169.770,52.477,160.188
C06216=1013.885,310.621,353.283,169.764,52.482,160.188
C06217=1013.879,310.373,353.316,169.758,52.488,160.188
C06218=1013.873,310.125,353.348,169.750,52.494,160.188
C06219=1013.867,309.877,353.381,169.744,52.500,160.188
C06220=1013.861,309.630,353.413,169.738,52.505,160.188
C06221=1013.855,309.382,353.445,169.732,52.511,160.188
C06222=1013.850,309.134,353.478,169.725,52.517,160.188
C06223=1013.843,308.886,353.509,169.718,52.523,160.188
C06224=1013.837,308.638,353.541,169.712,52.529,160.189
C06225=1013.829,308.352,353.578,169.705,52.535,160.189
C06226=1013.822,308.066,353.614,169.697,52.542,160.189
C06227=1013.816,307.781,353.651,169.689,52.550,160.189
C06228=1013.809,307.495,353.688,169.682,52.556,160.189
C06229=1013.802,307.247,353.719,169.677,52.563,160.189
C06230=1013.796,306.999,353.751,169.669,52.569,160.189
C06231=1013.790,306.751,353.782,169.663,52.575,160.189
C06232=1013.784,306.503,353.814,169.657,52.581,160.190
C06233=1013.777,306.255,353.846,169.651,52.587,160.190
C06234=1013.772,306.008,353.877,169.644,52.593,160.190
C06235=1013.765,305.760,353.909,169.638,52.599,160.190
C06236=1013.759,305.512,353.941,169.632,52.605,160.190
C06237=1013.753,305.264,353.972,169.625,52.612,160.190
C06238=1013.747,305.016,354.004,169.619,52.617,160.190
C06239=1013.741,304.768,354.034,169.612,52.623,160.190
C06240=1013.735,304.520,354.066,169.606,52.629,160.191
C06241=1013.729,304.272,354.098,169.599,52.635,160.191
C06242=1013.723,304.025,354.129,169.593,52.642,160.191
C06243=1013.717,303.777,354.161,169.587,52.647,160.191
C06244=1013.711,303.529,354.192,169.580,52.654,160.191
C06245=1013.705,303.281,354.224,169.574,52.660,160.191
C06246=1013.699,303.033,354.255,169.568,52.666,160.192
C06247=1013.693,302.784,354.286,169.562,52.673,160.192
C06248=1013.687,302.537,354.317,169.555,52.679,160.192
C06249=1013.681,302.289,354.349,169.549,52.685,160.192
C06250=1013.675,302.041,354.379,169.543,52.691,160.192
C06251=1013.670,301.793,354.412,169.537,52.697,160.193
C06252=1013.663,301.546,354.443,169.530,52.704,160.193
C06253=1013.658,301.297,354.474,169.524,52.710,160.193
C06254=1013.652,301.050,354.505,169.518,52.716,160.193
C06255=1013.646,300.802,354.537,169.513,52.723,160.194
C06256=1013.640,300.554,354.567,169.505,52.729,160.194
C06257=1013.634,300.306,354.599,169.500,52.735,160.194
C06258=1013.628,300.058,354.630,169.494,52.741,160.194
C06259=1013.623,299.810,354.661,169.488,52.748,160.194
C06260=1013.616,299.562,354.692,169.481,52.754,160.194
C06261=1013.611,299.314,354.724,169.475,52.760,160.195
C06262=1013.606,299.066,354.755,169.469,52.767,160.195
C06263=1013.599,298.818,354.785,169.462,52.774,160.195
C06264=1013.594,298.570,354.817,169.456,52.780,160.195
C06265=1013.588,298.322,354.847,169.450,52.786,160.196
C06266=1013.582,298.074,354.879,169.444,52.792,160.196
C06267=1013.576,297.826,354.910,169.438,52.799,160.196
C06268=1013.571,297.578,354.941,169.432,52.805,160.196
C06269=1013.564,297.330,354.972,169.426,52.812,160.197
C06270=1013.559,297.082,355.003,169.420,52.818,160.197
C06271=1013.554,296.834,355.033,169.413,52.825,160.197
C06272=1013.548,296.587,355.065,169.408,52.831,160.197
C06273=1013.542,296.338,355.096,169.401,52.837,160.197
C06274=1013.537,296.090,355.127,169.395,52.844,160.198
C06275=1013.531,295.842,355.157,169.389,52.850,160.198
C06276=1013.525,295.595,355.189,169.383,52.857,160.198
C06277=1013.519,295.346,355.220,169.377,52.863,160.199
C06278=1013.514,295.098,355.250,169.371,52.870,160.199
C06279=1013.508,294.850,355.281,169.364,52.876,160.199
C06280=1013.503,294.602,355.312,169.359,52.883,160.199
C06281=1013.497,294.355,355.343,169.353,52.889,160.200
C06282=1013.492,294.107,355.374,169.347,52.896,160.200
C06283=1013.485,293.858,355.404,169.341,52.903,160.200
C06284=1013.480,293.610,355.435,169.335,52.910,160.201
C06285=1013.475,293.342,355.468,169.328,52.916,160.201
C06286=1013.468,293.074,355.502,169.322,52.924,160.201
C06287=1013.463,292.806,355.535,169.315,52.931,160.201
C06288=1013.457,292.539,355.568,169.309,52.938,160.202
C06289=1013.451,292.291,355.599,169.303,52.945,160.202
C06290=1013.446,292.043,355.629,169.297,52.951,160.202
C06291=1013.440,291.795,355.659,169.292,52.958,160.203
C06292=1013.434,291.548,355.690,169.285,52.965,160.203
C06293=1013.428,291.299,355.719,169.279,52.971,160.203
C06294=1013.423,291.050,355.751,169.273,52.978,160.204
C06295=1013.417,290.803,355.781,169.267,52.985,160.204
C06296=1013.411,290.555,355.811,169.261,52.992,160.204
C06297=1013.406,290.306,355.841,169.256,52.999,160.205
C06298=1013.400,290.058,355.871,169.249,53.006,160.205
C06299=1013.394,289.811,355.902,169.243,53.012,160.205
C06300=1013.388,289.562,355.931,169.238,53.019,160.206
C06301=1013.383,289.314,355.962,169.231,53.026,160.206
C06302=1013.377,289.066,355.991,169.226,53.033,160.207
C06303=1013.371,288.818,356.022,169.220,53.040,160.207
C06304=1013.365,288.570,356.052,169.214,53.047,160.207
C06305=1013.360,288.322,356.082,169.208,53.054,160.208
C06306=1013.354,288.074,356.112,169.202,53.061,160.208
C06307=1013.349,287.826,356.142,169.196,53.067,160.208
C06308=1013.343,287.578,356.172,169.191,53.075,160.209
C06309=1013.338,287.330,356.201,169.184,53.081,160.209
C06310=1013.332,287.082,356.231,169.178,53.089,160.209
C06311=1013.327,286.834,356.261,169.173,53.096,160.210
C06312=1013.321,286.585,356.291,169.166,53.103,160.210
C06313=1013.315,286.338,356.321,169.161,53.110,160.211
C06314=1013.310,286.089,356.351,169.155,53.116,160.211
C06315=1013.304,285.841,356.380,169.149,53.124,160.211
C06316=1013.298,285.593,356.411,169.144,53.131,160.212
C06317=1013.293,285.344,356.440,169.137,53.138,160.212
C06318=1013.288,285.097,356.470,169.132,53.145,160.213
C06319=1013.282,284.849,356.500,169.126,53.152,160.213
C06320=1013.277,284.600,356.530,169.120,53.159,160.214
C06321=1013.271,284.352,356.559,169.114,53.166,160.214
C06322=1013.266,284.103,356.589,169.109,53.173,160.214
C06323=1013.259,283.856,356.619,169.102,53.181,160.215
C06324=1013.254,283.608,356.648,169.097,53.188,160.215
C06325=1013.249,283.360,356.678,169.091,53.195,160.216
C06326=1013.243,283.111,356.707,169.085,53.202,160.216
C06327=1013.237,282.863,356.736,169.079,53.209,160.216
C06328=1013.231,282.615,356.766,169.073,53.216,160.217
C06329=1013.226,282.367,356.795,169.068,53.224,160.217
C06330=1013.220,282.119,356.824,169.062,53.231,160.218
C06331=1013.215,281.870,356.854,169.057,53.238,160.218
C06332=1013.209,281.622,356.883,169.050,53.246,160.219
C06333=1013.204,281.374,356.913,169.045,53.253,160.219
C06334=1013.198,281.126,356.942,169.039,53.261,160.220
C06335=1013.193,280.878,356.971,169.033,53.268,160.220
C06336=1013.188,280.630,357.001,169.028,53.275,160.221
C06337=1013.181,280.382,357.030,169.022,53.282,160.221
C06338=1013.176,280.133,357.059,169.016,53.290,160.221
C06339=1013.171,279.884,357.088,169.010,53.297,160.222
C06340=1013.166,279.637,357.118,169.005,53.304,160.222
C06341=1013.159,279.388,357.147,168.998,53.312,160.223
C06342=1013.154,279.140,357.176,168.993,53.319,160.223
C06343=1013.149,278.892,357.205,168.988,53.326,160.224
C06344=1013.143,278.643,357.234,168.982,53.334,160.224
C06345=1013.138,278.388,357.264,168.976,53.342,160.225
C06346=1013.132,278.133,357.294,168.970,53.349,160.225
C06347=1013.127,277.877,357.325,168.964,53.357,160.226
C06348=1013.121,277.622,357.355,168.958,53.365,160.226
C06349=1013.116,277.373,357.383,168.953,53.372,160.227
C06350=1013.111,277.125,357.413,168.948,53.379,160.227
C06351=1013.104,276.877,357.442,168.941,53.387,160.228
C06352=1013.100,276.628,357.470,168.936,53.394,160.228
C06353=1013.094,276.380,357.500,168.930,53.402,160.229
C06354=1013.089,276.132,357.529,168.925,53.410,160.229
C06355=1013.083,275.883,357.558,168.919,53.417,160.230
C06356=1013.079,275.636,357.587,168.913,53.424,160.230
C06357=1013.072,275.387,357.616,168.908,53.433,160.231
C06358=1013.067,275.139,357.644,168.902,53.440,160.231
C06359=1013.062,274.890,357.673,168.896,53.447,160.232
C06360=1013.056,274.643,357.701,168.891,53.455,160.233
C06361=1013.051,274.394,357.730,168.885,53.463,160.233
C06362=1013.045,274.146,357.759,168.880,53.470,160.233
C06363=1013.040,273.897,357.788,168.874,53.478,160.234
C06364=1013.034,273.650,357.817,168.869,53.485,160.235
C06365=1013.029,273.401,357.846,168.863,53.494,160.235
C06366=1013.024,273.153,357.873,168.858,53.501,160.236
C06367=1013.018,272.904,357.903,168.852,53.509,160.236
C06368=1013.013,272.656,357.931,168.846,53.516,160.237
C06369=1013.008,272.408,357.959,168.840,53.524,160.237
C06370=1013.002,272.160,357.989,168.835,53.532,160.238
C06371=1012.997,271.912,358.017,168.829,53.539,160.238
C06372=1012.992,271.663,358.046,168.824,53.547,160.239
C06373=1012.983,271.319,358.085,168.816,53.558,160.240
C06374=1012.977,270.975,358.124,168.808,53.569,160.241
C06375=1012.970,270.631,358.164,168.801,53.580,160.241
C06376=1012.962,270.286,358.203,168.793,53.591,160.242
C06377=1012.768,273.436,357.478,168.831,53.604,160.253
C06378=1012.773,273.740,357.442,168.838,53.594,160.253
C06379=1012.780,274.045,357.407,168.844,53.585,160.252
C06380=1012.787,274.350,357.372,168.852,53.575,160.251
C06381=1012.794,274.654,357.337,168.858,53.566,160.250
C06382=1012.799,274.903,357.308,168.864,53.558,160.250
C06383=1012.805,275.151,357.279,168.871,53.550,160.250
C06384=1012.810,275.399,357.251,168.875,53.543,160.249
C06385=1012.816,275.647,357.222,168.882,53.535,160.249
C06386=1012.821,275.896,357.193,168.887,53.528,160.248
C06387=1012.827,276.144,357.164,168.893,53.519,160.247
C06388=1012.831,276.392,357.136,168.898,53.512,160.247
C06389=1012.837,276.641,357.106,168.904,53.505,160.247
C06390=1012.842,276.888,357.077,168.910,53.497,160.246
C06391=1012.848,277.137,357.048,168.915,53.489,160.245
C06392=1012.853,277.385,357.019,168.921,53.482,160.245
C06393=1012.858,277.633,356.989,168.927,53.474,160.245
C06394=1012.864,277.892,356.960,168.932,53.467,160.244
C06395=1012.869,278.148,356.930,168.938,53.459,160.243
C06396=1012.875,278.406,356.900,168.944,53.451,160.243
C06397=1012.880,278.664,356.869,168.950,53.443,160.242
C06398=1012.886,278.912,356.840,168.955,53.436,160.242
C06399=1012.892,279.161,356.811,168.962,53.428,160.241
C06400=1012.896,279.409,356.782,168.967,53.421,160.241
C06401=1012.902,279.658,356.752,168.973,53.414,160.241
C06402=1012.908,279.905,356.723,168.979,53.406,160.240
C06403=1012.913,280.154,356.694,168.985,53.399,160.240
C06404=1012.918,280.403,356.665,168.990,53.392,160.239
C06405=1012.924,280.650,356.636,168.996,53.384,160.239
C06406=1012.930,280.898,356.607,169.002,53.377,160.238
C06407=1012.935,281.147,356.577,169.008,53.369,160.238
C06408=1012.940,281.395,356.548,169.013,53.362,160.237
C06409=1012.946,281.643,356.519,169.020,53.355,160.237
C06410=1012.952,281.891,356.489,169.025,53.347,160.236
C06411=1012.957,282.140,356.459,169.031,53.340,160.236
C06412=1012.963,282.387,356.431,169.036,53.333,160.235
C06413=1012.968,282.636,356.402,169.043,53.325,160.235
C06414=1012.974,282.885,356.372,169.048,53.318,160.235
C06415=1012.980,283.133,356.343,169.054,53.310,160.234
C06416=1012.985,283.380,356.314,169.060,53.303,160.234
C06417=1012.990,283.629,356.284,169.066,53.296,160.234
C06418=1012.996,283.877,356.254,169.072,53.289,160.233
C06419=1013.002,284.125,356.225,169.077,53.282,160.232
C06420=1013.007,284.373,356.196,169.083,53.274,160.232
C06421=1013.013,284.621,356.166,169.089,53.267,160.232
C06422=1013.018,284.869,356.136,169.095,53.260,160.231
C06423=1013.024,285.117,356.106,169.101,53.253,160.231
C06424=1013.030,285.366,356.076,169.107,53.246,160.230
C06425=1013.034,285.613,356.047,169.112,53.239,160.230
C06426=1013.040,285.862,356.017,169.118,53.232,160.230
C06427=1013.046,286.110,355.987,169.124,53.225,160.229
C06428=1013.051,286.358,355.957,169.130,53.217,160.229
C06429=1013.057,286.607,355.928,169.136,53.210,160.229
C06430=1013.063,286.854,355.897,169.142,53.203,160.228
C06431=1013.068,287.103,355.868,169.148,53.196,160.228
C06432=1013.073,287.351,355.838,169.154,53.189,160.227
C06433=1013.079,287.598,355.808,169.159,53.182,160.227
C06434=1013.084,287.847,355.779,169.166,53.175,160.227
C06435=1013.090,288.095,355.748,169.171,53.168,160.226
C06436=1013.096,288.343,355.719,169.177,53.161,160.226
C06437=1013.102,288.591,355.688,169.183,53.154,160.225
C06438=1013.107,288.839,355.659,169.189,53.147,160.225
C06439=1013.113,289.087,355.628,169.195,53.140,160.225
C06440=1013.118,289.336,355.599,169.201,53.133,160.224
C06441=1013.124,289.584,355.568,169.207,53.126,160.224
C06442=1013.130,289.832,355.539,169.213,53.119,160.224
C06443=1013.136,290.080,355.508,169.219,53.113,160.223
C06444=1013.141,290.328,355.479,169.225,53.105,160.223
C06445=1013.147,290.576,355.448,169.231,53.099,160.223
C06446=1013.153,290.824,355.418,169.237,53.092,160.222
C06447=1013.158,291.072,355.387,169.243,53.085,160.222
C06448=1013.163,291.320,355.357,169.248,53.078,160.222
C06449=1013.169,291.568,355.327,169.255,53.071,160.221
C06450=1013.175,291.816,355.297,169.261,53.064,160.221
C06451=1013.181,292.064,355.266,169.267,53.057,160.221
C06452=1013.186,292.312,355.237,169.273,53.051,160.220
C06453=1013.191,292.560,355.206,169.278,53.044,160.220
C06454=1013.198,292.830,355.172,169.285,53.037,160.220
C06455=1013.204,293.100,355.139,169.292,53.030,160.219
C06456=1013.209,293.370,355.105,169.298,53.022,160.219
C06457=1013.215,293.641,355.072,169.305,53.015,160.219
C06458=1013.221,293.889,355.042,169.311,53.008,160.219
C06459=1013.226,294.136,355.010,169.317,53.002,160.218
C06460=1013.232,294.384,354.980,169.323,52.995,160.218
C06461=1013.238,294.633,354.948,169.329,52.988,160.218
C06462=1013.243,294.881,354.918,169.335,52.982,160.217
C06463=1013.249,295.129,354.887,169.341,52.975,160.217
C06464=1013.254,295.376,354.857,169.348,52.968,160.217
C06465=1013.259,295.625,354.826,169.354,52.962,160.217
C06466=1013.265,295.872,354.796,169.359,52.955,160.216
C06467=1013.271,296.121,354.763,169.366,52.949,160.216
C06468=1013.277,296.368,354.733,169.372,52.942,160.216
C06469=1013.282,296.617,354.702,169.378,52.936,160.215
C06470=1013.288,296.864,354.672,169.384,52.929,160.215
C06471=1013.293,297.112,354.640,169.390,52.923,160.215
C06472=1013.300,297.360,354.609,169.396,52.916,160.215
C06473=1013.305,297.609,354.579,169.403,52.909,160.214
C06474=1013.311,297.856,354.548,169.409,52.904,160.214
C06475=1013.316,298.104,354.517,169.415,52.897,160.214
C06476=1013.322,298.352,354.486,169.421,52.891,160.214
C06477=1013.328,298.601,354.455,169.427,52.884,160.214
C06478=1013.334,298.848,354.424,169.433,52.877,160.213
C06479=1013.339,299.097,354.392,169.439,52.871,160.213
C06480=1013.346,299.344,354.361,169.446,52.864,160.213
C06481=1013.351,299.592,354.330,169.452,52.859,160.213
C06482=1013.357,299.840,354.298,169.458,52.852,160.212
C06483=1013.362,300.088,354.268,169.465,52.845,160.212
C06484=1013.367,300.336,354.237,169.470,52.839,160.212
C06485=1013.374,300.584,354.206,169.476,52.832,160.212
C06486=1013.379,300.832,354.175,169.484,52.826,160.212
C06487=1013.386,301.080,354.143,169.489,52.820,160.211
C06488=1013.391,301.328,354.112,169.495,52.814,160.211
C06489=1013.397,301.575,354.081,169.502,52.807,160.211
C06490=1013.403,301.824,354.049,169.508,52.801,160.211
C06491=1013.409,302.071,354.019,169.514,52.795,160.211
C06492=1013.415,302.320,353.987,169.521,52.788,160.211
C06493=1013.421,302.567,353.957,169.527,52.782,160.210
C06494=1013.427,302.816,353.925,169.533,52.776,160.210
C06495=1013.433,303.063,353.893,169.540,52.770,160.210
C06496=1013.439,303.312,353.862,169.546,52.763,160.210
C06497=1013.445,303.559,353.831,169.552,52.757,160.209
C06498=1013.451,303.807,353.799,169.559,52.751,160.209
C06499=1013.457,304.054,353.768,169.565,52.744,160.209
C06500=1013.463,304.303,353.737,169.571,52.739,160.209
C06501=1013.469,304.550,353.706,169.578,52.732,160.209
C06502=1013.475,304.799,353.674,169.584,52.726,160.209
C06503=1013.481,305.046,353.643,169.590,52.720,160.209
C06504=1013.486,305.295,353.611,169.597,52.714,160.209
C06505=1013.492,305.543,353.579,169.603,52.707,160.208
C06506=1013.499,305.790,353.548,169.609,52.701,160.208
C06507=1013.505,306.038,353.516,169.616,52.695,160.208
C06508=1013.511,306.286,353.485,169.622,52.689,160.208
C06509=1013.517,306.534,353.453,169.628,52.683,160.208
C06510=1013.523,306.782,353.422,169.635,52.676,160.208
C06511=1013.529,307.030,353.390,169.642,52.671,160.208
C06512=1013.535,307.277,353.358,169.647,52.664,160.207
C06513=1013.541,307.526,353.327,169.655,52.658,160.207
C06514=1013.549,307.814,353.290,169.661,52.651,160.207
C06515=1013.556,308.102,353.253,169.669,52.644,160.207
C06516=1013.564,308.390,353.216,169.677,52.637,160.207
C06517=1013.570,308.679,353.180,169.685,52.630,160.207
C06518=1013.576,308.926,353.148,169.691,52.624,160.206
C06519=1013.583,309.173,353.116,169.697,52.618,160.206
C06520=1013.588,309.421,353.084,169.703,52.612,160.206
C06521=1013.594,309.669,353.051,169.710,52.606,160.206
C06522=1013.600,309.917,353.019,169.717,52.600,160.206
C06523=1013.606,310.165,352.987,169.723,52.595,160.206
C06524=1013.611,310.412,352.955,169.729,52.589,160.206
C06525=1013.617,310.660,352.923,169.736,52.583,160.206
C06526=1013.624,310.908,352.890,169.743,52.577,160.206
C06527=1013.629,311.156,352.857,169.749,52.572,160.206
C06528=1013.635,311.403,352.825,169.755,52.566,160.206
C06529=1013.641,311.651,352.792,169.763,52.560,160.206
C06530=1013.647,311.899,352.760,169.769,52.554,160.206
C06531=1013.653,312.147,352.727,169.775,52.548,160.206
C06532=1013.659,312.395,352.695,169.781,52.543,160.206
C06533=1013.664,312.642,352.662,169.789,52.537,160.206
C06534=1013.670,312.890,352.630,169.795,52.532,160.206
C06535=1013.676,313.138,352.598,169.802,52.526,160.206
C06536=1013.683,313.386,352.565,169.808,52.520,160.206
C06537=1013.689,313.633,352.532,169.815,52.514,160.206
C06538=1013.694,313.882,352.499,169.821,52.508,160.206
C06539=1013.701,314.129,352.467,169.828,52.503,160.206
C06540=1013.707,314.377,352.434,169.834,52.498,160.206
C06541=1013.713,314.624,352.401,169.842,52.492,160.206
C06542=1013.719,314.872,352.369,169.848,52.486,160.205
C06543=1013.725,315.120,352.337,169.854,52.480,160.205
C06544=1013.730,315.367,352.304,169.861,52.475,160.206
C06545=1013.737,315.615,352.271,169.868,52.469,160.206
C06546=1013.743,315.863,352.238,169.874,52.463,160.205
C06547=1013.749,316.110,352.205,169.881,52.458,160.206
C06548=1013.756,316.358,352.173,169.888,52.452,160.206
C06549=1013.762,316.606,352.139,169.895,52.447,160.206
C06550=1013.768,316.855,352.107,169.901,52.442,160.206
C06551=1013.774,317.102,352.074,169.908,52.436,160.206
C06552=1013.780,317.350,352.041,169.915,52.431,160.206
C06553=1013.787,317.597,352.009,169.922,52.425,160.206
C06554=1013.792,317.845,351.975,169.928,52.419,160.206
C06555=1013.798,318.093,351.942,169.935,52.414,160.206
C06556=1013.805,318.340,351.910,169.942,52.408,160.206
C06557=1013.811,318.588,351.877,169.948,52.403,160.206
C06558=1013.818,318.835,351.844,169.955,52.397,160.206
C06559=1013.824,319.083,351.810,169.962,52.392,160.206
C06560=1013.830,319.331,351.777,169.969,52.386,160.206
C06561=1013.836,319.579,351.744,169.975,52.381,160.206
C06562=1013.843,319.826,351.712,169.983,52.375,160.206
C06563=1013.849,320.074,351.679,169.989,52.370,160.206
C06564=1013.856,320.322,351.646,169.996,52.365,160.206
C06565=1013.862,320.570,351.612,170.003,52.359,160.206
C06566=1013.868,320.817,351.579,170.010,52.354,160.206
C06567=1013.874,321.065,351.546,170.016,52.349,160.206
C06568=1013.881,321.313,351.513,170.024,52.343,160.207
C06569=1013.888,321.560,351.480,170.031,52.338,160.207
C06570=1013.893,321.808,351.446,170.037,52.333,160.207
C06571=1013.900,322.056,351.413,170.045,52.327,160.207
C06572=1013.906,322.304,351.380,170.051,52.322,160.207
C06573=1013.913,322.551,351.347,170.058,52.317,160.207
C06574=1013.920,322.845,351.308,170.066,52.311,160.207
C06575=1013.928,323.138,351.268,170.075,52.304,160.207
C06576=1013.936,323.432,351.228,170.083,52.298,160.207
C06577=1013.944,323.726,351.189,170.091,52.291,160.208
C06578=1013.951,323.973,351.156,170.098,52.286,160.208
C06579=1013.956,324.221,351.122,170.105,52.281,160.208
C06580=1013.963,324.469,351.089,170.112,52.276,160.208
C06581=1013.970,324.716,351.056,170.119,52.271,160.208
C06582=1013.977,324.964,351.022,170.125,52.265,160.208
C06583=1013.983,325.211,350.989,170.133,52.260,160.208
C06584=1013.990,325.459,350.955,170.140,52.255,160.208
C06585=1013.996,325.706,350.921,170.148,52.250,160.209
C06586=1014.003,325.955,350.888,170.154,52.245,160.209
C06587=1014.009,326.202,350.854,170.161,52.240,160.209
C06588=1014.016,326.450,350.820,170.168,52.235,160.209
C06589=1014.022,326.697,350.786,170.176,52.230,160.209
C06590=1014.029,326.945,350.752,170.183,52.225,160.210
C06591=1014.034,327.192,350.718,170.189,52.220,160.210
C06592=1014.042,327.440,350.684,170.197,52.215,160.210
C06593=1014.048,327.688,350.650,170.204,52.210,160.210
C06594=1014.054,327.935,350.616,170.210,52.205,160.210
C06595=1014.061,328.183,350.582,170.219,52.200,160.211
C06596=1014.067,328.430,350.548,170.225,52.195,160.211
C06597=1014.074,328.678,350.513,170.232,52.190,160.211
C06598=1014.080,328.925,350.480,170.239,52.185,160.211
C06599=1014.087,329.173,350.445,170.247,52.180,160.211
C06600=1014.093,329.421,350.411,170.254,52.175,160.211
C06601=1014.100,329.668,350.378,170.260,52.170,160.212
C06602=1014.106,329.916,350.343,170.268,52.166,160.212
C06603=1014.113,330.164,350.309,170.275,52.161,160.212
C06604=1014.120,330.412,350.275,170.282,52.156,160.212
C06605=1014.126,330.658,350.240,170.290,52.151,160.213
C06606=1014.132,330.906,350.206,170.297,52.146,160.213
C06607=1014.140,331.154,350.172,170.303,52.141,160.213
C06608=1014.145,331.401,350.138,170.312,52.136,160.213
C06609=1014.152,331.649,350.103,170.318,52.131,160.213
C06610=1014.159,331.896,350.069,170.325,52.127,160.214
C06611=1014.166,332.144,350.034,170.333,52.122,160.214
C06612=1014.173,332.392,349.999,170.340,52.117,160.214
C06613=1014.179,332.639,349.965,170.347,52.112,160.214
C06614=1014.185,332.886,349.930,170.355,52.108,160.215
C06615=1014.192,333.134,349.896,170.362,52.103,160.215
C06616=1014.199,333.382,349.861,170.369,52.098,160.215
C06617=1014.206,333.629,349.827,170.377,52.094,160.216
C06618=1014.212,333.876,349.792,170.384,52.089,160.216
C06619=1014.218,334.124,349.758,170.391,52.084,160.216
C06620=1014.225,334.371,349.722,170.399,52.080,160.217
C06621=1014.232,334.619,349.687,170.406,52.075,160.217
C06622=1014.238,334.867,349.653,170.413,52.070,160.217
C06623=1014.245,335.114,349.618,170.421,52.066,160.218
C06624=1014.252,335.361,349.583,170.428,52.061,160.218
C06625=1014.258,335.609,349.548,170.435,52.057,160.218
C06626=1014.265,335.857,349.513,170.443,52.052,160.218
C06627=1014.272,336.104,349.478,170.450,52.047,160.219
C06628=1014.279,336.352,349.443,170.458,52.043,160.219
C06629=1014.286,336.599,349.409,170.466,52.038,160.220
C06630=1014.293,336.847,349.374,170.473,52.034,160.220
C06631=1014.299,337.094,349.339,170.481,52.029,160.220
C06632=1014.306,337.341,349.304,170.488,52.025,160.221
C06633=1014.313,337.589,349.268,170.495,52.021,160.221
C06634=1014.321,337.878,349.227,170.504,52.015,160.221
C06635=1014.329,338.168,349.186,170.513,52.010,160.222
C06636=1014.336,338.456,349.145,170.522,52.004,160.222
C06637=1014.344,338.746,349.104,170.531,51.999,160.223
C06638=1014.351,338.994,349.069,170.538,51.995,160.223
C06639=1014.358,339.241,349.034,170.545,51.990,160.223
C06640=1014.365,339.488,348.999,170.553,51.986,160.224
C06641=1014.372,339.736,348.962,170.561,51.982,160.224
C06642=1014.378,339.983,348.927,170.569,51.977,160.225
C06643=1014.385,340.231,348.891,170.576,51.973,160.225
C06644=1014.392,340.478,348.856,170.583,51.969,160.225
C06645=1014.399,340.725,348.820,170.591,51.964,160.226
C06646=1014.406,340.973,348.785,170.599,51.960,160.226
C06647=1014.412,341.221,348.749,170.607,51.956,160.227
C06648=1014.420,341.467,348.713,170.614,51.951,160.227
C06649=1014.426,341.715,348.678,170.621,51.947,160.227
C06650=1014.434,341.963,348.643,170.630,51.943,160.228
C06651=1014.441,342.210,348.607,170.637,51.939,160.228
C06652=1014.447,342.457,348.571,170.645,51.934,160.229
C06653=1014.454,342.704,348.535,170.653,51.931,160.229
C06654=1014.461,342.952,348.500,170.660,51.926,160.230
C06655=1014.468,343.199,348.464,170.669,51.922,160.230
C06656=1014.474,343.446,348.428,170.676,51.918,160.231
C06657=1014.482,343.694,348.392,170.684,51.913,160.231
C06658=1014.489,343.941,348.357,170.691,51.910,160.232
C06659=1014.496,344.188,348.321,170.700,51.905,160.232
C06660=1014.503,344.436,348.284,170.707,51.901,160.233
C06661=1014.510,344.683,348.249,170.714,51.897,160.233
C06662=1014.517,344.931,348.213,170.723,51.893,160.233
C06663=1014.524,345.178,348.176,170.730,51.889,160.234
C06664=1014.531,345.426,348.141,170.739,51.885,160.234
C06665=1014.538,345.672,348.105,170.746,51.881,160.235
C06666=1014.546,345.920,348.069,170.754,51.876,160.235
C06667=1014.552,346.167,348.032,170.762,51.873,160.236
C06668=1014.560,346.414,347.996,170.770,51.869,160.237
C06669=1014.567,346.661,347.960,170.778,51.864,160.237
C06670=1014.574,346.909,347.924,170.786,51.860,160.238
C06671=1014.581,347.156,347.888,170.794,51.857,160.238
C06672=1014.588,347.403,347.851,170.802,51.853,160.239
C06673=1014.595,347.650,347.815,170.809,51.848,160.239
C06674=1014.602,347.898,347.778,170.818,51.844,160.240
C06675=1014.609,348.145,347.742,170.826,51.841,160.240
C06676=1014.616,348.392,347.706,170.834,51.837,160.241
C06677=1014.623,348.640,347.669,170.842,51.833,160.241
C06678=1014.630,348.887,347.633,170.850,51.829,160.242
C06679=1014.637,349.134,347.597,170.858,51.825,160.243
C06680=1014.644,349.381,347.560,170.866,51.821,160.243
C06681=1014.652,349.628,347.523,170.874,51.818,160.244
C06682=1014.659,349.876,347.486,170.883,51.813,160.244
C06683=1014.666,350.123,347.451,170.890,51.810,160.245
C06684=1014.673,350.370,347.413,170.899,51.806,160.246
C06685=1014.680,350.618,347.376,170.906,51.802,160.246
C06686=1014.688,350.865,347.340,170.915,51.798,160.247
C06687=1014.694,351.111,347.303,170.922,51.794,160.247
C06688=1014.702,351.359,347.267,170.931,51.790,160.248
C06689=1014.709,351.606,347.229,170.939,51.787,160.248
C06690=1014.717,351.853,347.193,170.947,51.783,160.249
C06691=1014.724,352.101,347.155,170.955,51.779,160.250
C06692=1014.731,352.347,347.120,170.963,51.775,160.250
C06693=1014.738,352.594,347.082,170.972,51.772,160.251
C06694=1014.747,352.881,347.040,170.981,51.768,160.252
C06695=1014.756,353.168,346.997,170.990,51.763,160.252
C06696=1014.764,353.455,346.954,171.000,51.759,160.253
C06697=1014.773,353.742,346.911,171.010,51.755,160.254
C06698=1014.780,353.989,346.874,171.019,51.751,160.255
C06699=1014.788,354.236,346.836,171.026,51.748,160.255
C06700=1014.794,354.482,346.799,171.035,51.743,160.256
C06701=1014.801,354.730,346.762,171.044,51.740,160.257
C06702=1014.809,354.977,346.725,171.051,51.736,160.257
C06703=1014.817,355.224,346.688,171.060,51.733,160.258
C06704=1014.824,355.471,346.650,171.068,51.729,160.259
C06705=1014.831,355.718,346.613,171.077,51.726,160.259
C06706=1014.839,355.965,346.576,171.085,51.722,160.260
C06707=1014.846,356.212,346.538,171.093,51.719,160.261
C06708=1014.854,356.459,346.501,171.102,51.715,160.261
C06709=1014.861,356.706,346.464,171.111,51.712,160.262
C06710=1014.869,356.954,346.426,171.119,51.709,160.263
C06711=1014.877,357.201,346.388,171.127,51.705,160.264
C06712=1014.884,357.448,346.351,171.136,51.701,160.264
C06713=1014.891,357.696,346.313,171.144,51.698,160.265
C06714=1014.899,357.942,346.276,171.153,51.694,160.266
C06715=1014.907,358.189,346.238,171.162,51.691,160.267
C06716=1014.914,358.436,346.201,171.170,51.688,160.267
C06717=1014.922,358.684,346.163,171.178,51.684,160.268
C06718=1014.929,358.930,346.125,171.187,51.680,160.269
C06719=1014.936,359.177,346.087,171.195,51.677,160.270
C06720=1014.944,359.425,346.050,171.204,51.674,160.271
C06721=1014.951,359.671,346.011,171.213,51.671,160.271
C06722=1014.959,359.918,345.974,171.221,51.668,160.272
C06723=1014.967,360.165,345.935,171.230,51.664,160.273
C06724=1014.974,360.413,345.898,171.239,51.661,160.274
C06725=1014.981,360.659,345.859,171.247,51.658,160.275
C06726=1014.989,360.906,345.821,171.256,51.655,160.275
C06727=1014.997,361.153,345.783,171.265,51.651,160.276
C06728=1015.004,361.400,345.745,171.273,51.648,160.277
C06729=1015.012,361.647,345.707,171.282,51.645,160.278
C06730=1015.020,361.894,345.669,171.291,51.641,160.279
C06731=1015.027,362.141,345.631,171.300,51.638,160.279
C06732=1015.036,362.388,345.592,171.308,51.635,160.280
C06733=1015.043,362.635,345.554,171.317,51.632,160.281
C06734=1015.050,362.882,345.516,171.327,51.629,160.282
C06735=1015.058,363.129,345.477,171.336,51.625,160.283
C06736=1015.065,363.376,345.439,171.344,51.622,160.284
C06737=1015.073,363.623,345.400,171.353,51.619,160.284
C06738=1015.081,363.870,345.362,171.362,51.616,160.286
C06739=1015.089,364.117,345.323,171.371,51.613,160.286
C06740=1015.097,364.363,345.285,171.380,51.610,160.287
C06741=1015.105,364.610,345.246,171.388,51.607,160.288
C06742=1015.112,364.857,345.208,171.397,51.604,160.289
C06743=1015.121,365.104,345.170,171.406,51.600,160.290
C06744=1015.128,365.351,345.131,171.416,51.598,160.291
C06745=1015.136,365.598,345.093,171.425,51.594,160.292
C06746=1015.144,365.845,345.054,171.434,51.592,160.293
C06747=1015.152,366.092,345.016,171.442,51.589,160.294
C06748=1015.160,366.339,344.977,171.451,51.585,160.294
C06749=1015.168,366.585,344.938,171.460,51.582,160.295
C06750=1015.176,366.832,344.900,171.470,51.580,160.296
C06751=1015.184,367.079,344.861,171.479,51.576,160.297
C06752=1015.191,367.326,344.822,171.488,51.574,160.298
C06753=1015.199,367.573,344.783,171.497,51.570,160.299
C06754=1015.208,367.867,344.737,171.508,51.567,160.300
C06755=1015.218,368.161,344.690,171.519,51.564,160.302
C06756=1015.228,368.456,344.643,171.529,51.560,160.303
C06757=1015.237,368.750,344.597,171.541,51.557,160.304
C06758=1015.245,368.997,344.557,171.550,51.554,160.305
C06759=1015.253,369.243,344.518,171.559,51.551,160.306
C06760=1015.261,369.490,344.479,171.569,51.549,160.307
C06761=1015.268,369.737,344.439,171.578,51.545,160.308
C06762=1015.277,369.984,344.400,171.587,51.543,160.309
C06763=1015.285,370.231,344.361,171.596,51.540,160.310
C06764=1015.293,370.478,344.321,171.605,51.537,160.311
C06765=1015.301,370.724,344.282,171.614,51.535,160.312
C06766=1015.308,370.971,344.242,171.624,51.532,160.313
C06767=1015.317,371.217,344.203,171.633,51.529,160.314
C06768=1015.325,371.464,344.164,171.643,51.526,160.315
C06769=1015.333,371.711,344.124,171.652,51.524,160.316
C06770=1015.341,371.957,344.085,171.661,51.521,160.317
C06771=1015.350,372.204,344.045,171.671,51.519,160.318
C06772=1015.358,372.451,344.005,171.681,51.516,160.320
C06773=1015.366,372.697,343.966,171.690,51.513,160.321
C06774=1015.374,372.944,343.926,171.699,51.510,160.322
C06775=1015.382,373.191,343.887,171.709,51.508,160.323
C06776=1015.391,373.438,343.847,171.719,51.505,160.324
C06777=1015.398,373.684,343.807,171.729,51.502,160.325
C06778=1015.407,373.931,343.768,171.738,51.500,160.326
C06779=1015.415,374.179,343.728,171.748,51.497,160.327
C06780=1015.424,374.425,343.688,171.758,51.495,160.328
C06781=1015.432,374.671,343.648,171.767,51.492,160.329
C06782=1015.440,374.918,343.609,171.776,51.489,160.330
C06783=1015.449,375.164,343.569,171.786,51.487,160.332
C06784=1015.458,375.411,343.529,171.795,51.484,160.333
C06785=1015.466,375.658,343.489,171.805,51.482,160.334
C06786=1015.474,375.905,343.448,171.816,51.479,160.335
C06787=1015.482,376.151,343.408,171.825,51.477,160.336
C06788=1015.490,376.397,343.368,171.835,51.475,160.338
C06789=1015.499,376.644,343.327,171.845,51.472,160.339
C06790=1015.507,376.891,343.287,171.854,51.470,160.340
C06791=1015.515,377.138,343.247,171.864,51.468,160.341
C06792=1015.523,377.384,343.207,171.874,51.465,160.342
C06793=1015.532,377.631,343.166,171.884,51.463,160.344
C06794=1015.540,377.877,343.125,171.894,51.460,160.345
C06795=1015.549,378.123,343.085,171.904,51.458,160.346
C06796=1015.557,378.370,343.045,171.913,51.456,160.347
C06797=1015.565,378.617,343.004,171.923,51.453,160.348
C06798=1015.574,378.864,342.963,171.934,51.451,160.350
C06799=1015.583,379.110,342.923,171.944,51.449,160.351
C06800=1015.591,379.356,342.882,171.954,51.447,160.352
C06801=1015.599,379.603,342.841,171.963,51.444,160.354
C06802=1015.607,379.849,342.801,171.974,51.442,160.355
C06803=1015.617,380.096,342.760,171.984,51.440,160.356
C06804=1015.625,380.342,342.719,171.994,51.438,160.357
C06805=1015.634,380.589,342.678,172.004,51.435,160.359
C06806=1015.642,380.835,342.638,172.014,51.433,160.360
C06807=1015.651,381.082,342.597,172.024,51.431,160.361
C06808=1015.660,381.329,342.556,172.034,51.429,160.363
C06809=1015.668,381.574,342.515,172.045,51.426,160.364
C06810=1015.677,381.821,342.474,172.055,51.424,160.365
C06811=1015.686,382.068,342.433,172.065,51.422,160.367
C06812=1015.694,382.313,342.392,172.076,51.420,160.368
C06813=1015.704,382.560,342.352,172.085,51.418,160.369
C06814=1015.714,382.878,342.298,172.099,51.415,160.371
C06815=1015.725,383.194,342.245,172.112,51.412,160.373
C06816=1015.737,383.511,342.193,172.125,51.410,160.374
C06817=1015.749,383.828,342.140,172.139,51.407,160.376
C06818=1015.757,384.075,342.099,172.149,51.405,160.378
C06819=1015.767,384.321,342.057,172.159,51.403,160.379
C06820=1015.776,384.568,342.016,172.170,51.401,160.380
C06821=1015.784,384.814,341.975,172.180,51.399,160.382
C06822=1015.793,385.060,341.933,172.191,51.396,160.383
C06823=1015.802,385.306,341.892,172.201,51.395,160.385
C06824=1015.811,385.553,341.850,172.212,51.393,160.386
C06825=1015.820,385.799,341.808,172.222,51.391,160.387
C06826=1015.829,386.045,341.767,172.233,51.389,160.389
C06827=1015.837,386.292,341.725,172.244,51.387,160.391
C06828=1015.846,386.538,341.683,172.255,51.385,160.392
C06829=1015.855,386.784,341.641,172.264,51.383,160.393
C06830=1015.864,387.031,341.600,172.276,51.381,160.395
C06831=1015.873,387.277,341.558,172.287,51.379,160.396
C06832=1015.882,387.524,341.516,172.297,51.378,160.398
C06833=1015.891,387.770,341.475,172.308,51.376,160.399
C06834=1015.900,388.016,341.432,172.319,51.374,160.401
C06835=1015.909,388.262,341.390,172.330,51.373,160.403
C06836=1015.918,388.508,341.349,172.340,51.371,160.404
C06837=1015.927,388.754,341.306,172.351,51.369,160.406
C06838=1015.936,389.001,341.265,172.362,51.367,160.407
C06839=1015.946,389.246,341.222,172.373,51.366,160.409
C06840=1015.954,389.493,341.180,172.384,51.364,160.410
C06841=1015.964,389.739,341.137,172.395,51.362,160.412
C06842=1015.973,389.986,341.095,172.405,51.360,160.413
C06843=1015.982,390.231,341.053,172.417,51.359,160.415
C06844=1015.991,390.478,341.011,172.428,51.357,160.416
C06845=1016.001,390.724,340.968,172.439,51.355,160.418
C06846=1016.010,390.970,340.926,172.449,51.353,160.419
C06847=1016.019,391.216,340.884,172.461,51.352,160.421
C06848=1016.027,391.462,340.841,172.472,51.350,160.423
C06849=1016.037,391.709,340.798,172.483,51.348,160.424
C06850=1016.046,391.955,340.756,172.494,51.347,160.426
C06851=1016.056,392.201,340.713,172.505,51.345,160.428
C06852=1016.065,392.447,340.670,172.517,51.344,160.429
C06853=1016.074,392.693,340.628,172.528,51.342,160.431
C06854=1016.084,392.939,340.585,172.538,51.341,160.433
C06855=1016.093,393.185,340.542,172.550,51.340,160.434
C06856=1016.102,393.432,340.499,172.561,51.338,160.436
C06857=1016.111,393.678,340.457,172.573,51.336,160.438
C06858=1016.121,393.924,340.414,172.585,51.335,160.440
C06859=1016.130,394.169,340.370,172.596,51.333,160.441
C06860=1016.140,394.416,340.327,172.607,51.332,160.443
C06861=1016.149,394.662,340.285,172.619,51.331,160.445
C06862=1016.158,394.908,340.241,172.630,51.330,160.446
C06863=1016.168,395.154,340.198,172.641,51.328,160.448
C06864=1016.178,395.400,340.155,172.652,51.326,160.450
C06865=1016.188,395.646,340.112,172.664,51.325,160.451
C06866=1016.196,395.892,340.069,172.675,51.324,160.453
C06867=1016.206,396.138,340.025,172.687,51.322,160.455
C06868=1016.216,396.384,339.983,172.699,51.321,160.457
C06869=1016.226,396.630,339.939,172.710,51.319,160.459
C06870=1016.235,396.876,339.896,172.722,51.318,160.460
C06871=1016.244,397.122,339.852,172.733,51.317,160.462
C06872=1016.254,397.368,339.808,172.746,51.316,160.464
C06873=1016.265,397.614,339.765,172.757,51.315,160.466
C06874=1016.275,397.892,339.716,172.771,51.313,160.468
C06875=1016.286,398.169,339.666,172.784,51.311,160.470
C06876=1016.297,398.446,339.617,172.798,51.310,160.472
C06877=1016.308,398.724,339.568,172.811,51.309,160.474
C06878=1016.318,398.969,339.524,172.823,51.308,160.476
C06879=1016.327,399.216,339.480,172.834,51.307,160.478
C06880=1016.337,399.461,339.437,172.846,51.305,160.480
C06881=1016.346,399.707,339.393,172.859,51.304,160.482
C06882=1016.356,399.953,339.349,172.870,51.303,160.483
C06883=1016.366,400.198,339.304,172.882,51.302,160.485
C06884=1016.375,400.444,339.260,172.895,51.301,160.487
C06885=1016.386,400.691,339.216,172.906,51.300,160.489
C06886=1016.396,400.936,339.172,172.919,51.299,160.491
C06887=1016.405,401.182,339.127,172.931,51.298,160.493
C06888=1016.415,401.428,339.083,172.943,51.297,160.495
C06889=1016.425,401.674,339.039,172.955,51.296,160.497
C06890=1016.435,401.919,338.994,172.968,51.295,160.499
C06891=1016.444,402.165,338.950,172.980,51.294,160.501
C06892=1016.455,402.411,338.906,172.992,51.293,160.503
C06893=1016.464,402.656,338.861,173.005,51.292,160.505
C06894=1016.108,400.645,338.881,172.888,51.366,160.504
C06895=1016.098,400.399,338.925,172.876,51.367,160.502
C06896=1016.088,400.153,338.968,172.863,51.368,160.500
C06897=1016.079,399.908,339.013,172.852,51.370,160.498
C06898=1016.068,399.662,339.057,172.840,51.370,160.496
C06899=1016.059,399.416,339.101,172.828,51.372,160.495
C06900=1016.049,399.171,339.145,172.816,51.374,160.493
C06901=1016.040,398.926,339.188,172.804,51.374,160.491
C06902=1016.029,398.680,339.231,172.792,51.376,160.489
C06903=1016.020,398.436,339.276,172.780,51.377,160.487
C06904=1016.011,398.191,339.319,172.768,51.378,160.485
C06905=1016.001,397.945,339.362,172.757,51.379,160.483
C06906=1015.992,397.700,339.405,172.744,51.381,160.481
C06907=1015.982,397.454,339.449,172.733,51.382,160.480
C06908=1015.972,397.208,339.493,172.721,51.384,160.478
C06909=1015.962,396.963,339.536,172.709,51.385,160.476
C06910=1015.953,396.716,339.579,172.698,51.386,160.474
C06911=1015.943,396.471,339.623,172.686,51.388,160.473
C06912=1015.934,396.224,339.666,172.675,51.389,160.471
C06913=1015.924,395.978,339.710,172.663,51.391,160.469
C06914=1015.915,395.732,339.752,172.651,51.392,160.467
C06915=1015.905,395.487,339.796,172.640,51.393,160.465
C06916=1015.896,395.240,339.839,172.629,51.395,160.464
C06917=1015.886,394.994,339.882,172.617,51.397,160.462
C06918=1015.876,394.748,339.925,172.605,51.398,160.460
C06919=1015.868,394.502,339.968,172.594,51.399,160.459
C06920=1015.858,394.256,340.011,172.583,51.401,160.457
C06921=1015.848,394.011,340.054,172.571,51.403,160.455
C06922=1015.839,393.764,340.098,172.559,51.404,160.453
C06923=1015.830,393.518,340.140,172.548,51.406,160.452
C06924=1015.820,393.272,340.183,172.537,51.407,160.450
C06925=1015.811,393.026,340.225,172.525,51.409,160.449
C06926=1015.802,392.779,340.269,172.514,51.411,160.447
C06927=1015.793,392.533,340.311,172.503,51.413,160.445
C06928=1015.783,392.288,340.353,172.492,51.413,160.443
C06929=1015.774,392.041,340.397,172.481,51.415,160.442
C06930=1015.765,391.795,340.439,172.470,51.417,160.440
C06931=1015.756,391.549,340.482,172.458,51.419,160.439
C06932=1015.746,391.302,340.524,172.447,51.421,160.437
C06933=1015.737,391.057,340.566,172.436,51.423,160.435
C06934=1015.728,390.811,340.609,172.425,51.424,160.434
C06935=1015.720,390.564,340.651,172.414,51.426,160.432
C06936=1015.710,390.318,340.694,172.403,51.427,160.431
C06937=1015.700,390.072,340.736,172.391,51.429,160.429
C06938=1015.691,389.826,340.778,172.380,51.431,160.428
C06939=1015.682,389.580,340.820,172.370,51.433,160.426
C06940=1015.673,389.334,340.862,172.359,51.435,160.424
C06941=1015.663,389.087,340.905,172.348,51.437,160.423
C06942=1015.655,388.841,340.947,172.337,51.438,160.421
C06943=1015.646,388.594,340.988,172.326,51.440,160.420
C06944=1015.637,388.348,341.031,172.315,51.442,160.418
C06945=1015.628,388.102,341.073,172.305,51.444,160.417
C06946=1015.619,387.856,341.115,172.294,51.446,160.415
C06947=1015.610,387.609,341.156,172.282,51.448,160.414
C06948=1015.601,387.363,341.199,172.272,51.449,160.412
C06949=1015.592,387.117,341.241,172.261,51.452,160.411
C06950=1015.583,386.871,341.282,172.250,51.454,160.409
C06951=1015.574,386.624,341.324,172.240,51.455,160.408
C06952=1015.565,386.378,341.366,172.229,51.458,160.406
C06953=1015.556,386.132,341.407,172.219,51.459,160.405
C06954=1015.547,385.885,341.449,172.208,51.461,160.403
C06955=1015.539,385.639,341.491,172.197,51.464,160.402
C06956=1015.530,385.393,341.533,172.187,51.465,160.401
C06957=1015.522,385.146,341.573,172.176,51.468,160.399
C06958=1015.513,384.900,341.615,172.166,51.470,160.398
C06959=1015.504,384.654,341.657,172.155,51.472,160.396
C06960=1015.494,384.407,341.698,172.145,51.474,160.395
C06961=1015.485,384.160,341.739,172.134,51.476,160.394
C06962=1015.476,383.914,341.781,172.124,51.478,160.392
C06963=1015.465,383.595,341.833,172.110,51.481,160.391
C06964=1015.454,383.275,341.887,172.097,51.484,160.389
C06965=1015.443,382.957,341.940,172.084,51.487,160.387
C06966=1015.431,382.637,341.993,172.069,51.490,160.385
C06967=1015.422,382.390,342.034,172.060,51.492,160.384
C06968=1015.414,382.144,342.074,172.050,51.494,160.383
C06969=1015.405,381.898,342.116,172.039,51.496,160.381
C06970=1015.396,381.651,342.157,172.029,51.498,160.380
C06971=1015.387,381.405,342.197,172.018,51.501,160.378
C06972=1015.379,381.158,342.238,172.008,51.503,160.377
C06973=1015.370,380.912,342.279,171.997,51.505,160.376
C06974=1015.361,380.666,342.320,171.988,51.508,160.375
C06975=1015.353,380.419,342.360,171.978,51.510,160.373
C06976=1015.344,380.172,342.401,171.967,51.512,160.372
C06977=1015.336,379.926,342.442,171.957,51.514,160.371
C06978=1015.327,379.679,342.482,171.948,51.517,160.370
C06979=1015.319,379.433,342.523,171.937,51.520,160.368
C06980=1015.310,379.186,342.564,171.927,51.522,160.367
C06981=1015.302,378.940,342.605,171.917,51.524,160.366
C06982=1015.293,378.694,342.645,171.907,51.527,160.364
C06983=1015.285,378.447,342.686,171.897,51.529,160.363
C06984=1015.277,378.201,342.726,171.887,51.531,160.362
C06985=1015.268,377.953,342.766,171.878,51.534,160.361
C06986=1015.260,377.707,342.807,171.867,51.536,160.360
C06987=1015.252,377.461,342.847,171.857,51.539,160.358
C06988=1015.244,377.215,342.888,171.848,51.541,160.357
C06989=1015.235,376.967,342.928,171.838,51.544,160.356
C06990=1015.227,376.721,342.968,171.827,51.546,160.355
C06991=1015.219,376.475,343.009,171.818,51.549,160.354
C06992=1015.210,376.228,343.048,171.808,51.551,160.353
C06993=1015.201,375.981,343.089,171.798,51.553,160.351
C06994=1015.193,375.735,343.130,171.789,51.556,160.350
C06995=1015.186,375.488,343.170,171.779,51.558,160.349
C06996=1015.177,375.242,343.210,171.769,51.562,160.348
C06997=1015.169,374.995,343.250,171.760,51.564,160.347
C06998=1015.160,374.748,343.289,171.750,51.566,160.345
C06999=1015.152,374.501,343.329,171.740,51.569,160.344
C07000=1015.144,374.255,343.369,171.731,51.572,160.343
C07001=1015.135,374.008,343.409,171.721,51.575,160.342
C07002=1015.127,373.762,343.448,171.711,51.577,160.341
C07003=1015.119,373.515,343.488,171.701,51.580,160.340
C07004=1015.111,373.268,343.527,171.692,51.583,160.339
C07005=1015.103,373.021,343.567,171.683,51.586,160.338
C07006=1015.094,372.775,343.607,171.673,51.588,160.337
C07007=1015.086,372.528,343.646,171.664,51.591,160.336
C07008=1015.078,372.281,343.686,171.654,51.594,160.335
C07009=1015.070,372.035,343.725,171.645,51.597,160.334
C07010=1015.062,371.788,343.765,171.635,51.600,160.332
C07011=1015.054,371.541,343.804,171.625,51.603,160.331
C07012=1015.045,371.294,343.844,171.616,51.605,160.330
C07013=1015.037,371.048,343.884,171.606,51.608,160.329
C07014=1015.029,370.801,343.923,171.597,51.611,160.328
C07015=1015.021,370.554,343.962,171.588,51.614,160.327
C07016=1015.013,370.307,344.001,171.578,51.616,160.326
C07017=1015.005,370.061,344.040,171.569,51.619,160.325
C07018=1014.998,369.814,344.080,171.559,51.622,160.324
C07019=1014.989,369.567,344.119,171.551,51.625,160.323
C07020=1014.981,369.320,344.158,171.541,51.628,160.322
C07021=1014.973,369.073,344.198,171.532,51.631,160.321
C07022=1014.966,368.827,344.236,171.522,51.634,160.320
C07023=1014.956,368.530,344.284,171.511,51.637,160.319
C07024=1014.947,368.234,344.330,171.501,51.641,160.318
C07025=1014.937,367.937,344.378,171.490,51.644,160.317
C07026=1014.928,367.640,344.425,171.478,51.648,160.315
C07027=1014.920,367.393,344.464,171.469,51.651,160.314
C07028=1014.912,367.147,344.503,171.460,51.654,160.314
C07029=1014.904,366.900,344.541,171.450,51.657,160.312
C07030=1014.896,366.653,344.580,171.441,51.660,160.312
C07031=1014.889,366.406,344.619,171.433,51.663,160.311
C07032=1014.881,366.160,344.658,171.424,51.666,160.310
C07033=1014.873,365.913,344.696,171.415,51.669,160.309
C07034=1014.865,365.666,344.735,171.406,51.672,160.308
C07035=1014.857,365.419,344.773,171.397,51.676,160.307
C07036=1014.849,365.172,344.812,171.388,51.679,160.306
C07037=1014.841,364.925,344.850,171.378,51.682,160.305
C07038=1014.833,364.678,344.888,171.369,51.685,160.304
C07039=1014.825,364.431,344.927,171.360,51.688,160.304
C07040=1014.818,364.185,344.965,171.351,51.692,160.303
C07041=1014.810,363.937,345.004,171.343,51.694,160.302
C07042=1014.802,363.691,345.042,171.334,51.698,160.301
C07043=1014.794,363.443,345.080,171.325,51.701,160.300
C07044=1014.787,363.197,345.118,171.316,51.704,160.299
C07045=1014.779,362.950,345.157,171.307,51.708,160.298
C07046=1014.771,362.703,345.195,171.298,51.711,160.298
C07047=1014.763,362.456,345.233,171.289,51.714,160.296
C07048=1014.756,362.208,345.271,171.281,51.717,160.296
C07049=1014.748,361.962,345.310,171.272,51.720,160.295
C07050=1014.740,361.715,345.348,171.263,51.724,160.294
C07051=1014.733,361.468,345.386,171.254,51.727,160.293
C07052=1014.726,361.221,345.425,171.245,51.731,160.292
C07053=1014.718,360.974,345.463,171.237,51.734,160.292
C07054=1014.711,360.727,345.500,171.228,51.737,160.291
C07055=1014.703,360.480,345.539,171.219,51.741,160.290
C07056=1014.696,360.233,345.576,171.210,51.744,160.289
C07057=1014.688,359.986,345.615,171.202,51.747,160.289
C07058=1014.681,359.739,345.652,171.193,51.751,160.288
C07059=1014.673,359.492,345.691,171.184,51.754,160.287
C07060=1014.665,359.245,345.728,171.175,51.758,160.286
C07061=1014.658,358.998,345.766,171.168,51.761,160.286
C07062=1014.651,358.751,345.804,171.159,51.765,160.285
C07063=1014.643,358.504,345.842,171.150,51.768,160.284
C07064=1014.636,358.257,345.879,171.141,51.771,160.283
C07065=1014.628,358.010,345.916,171.133,51.775,160.282
C07066=1014.620,357.762,345.954,171.124,51.778,160.282
C07067=1014.613,357.516,345.992,171.116,51.783,160.281
C07068=1014.606,357.269,346.030,171.108,51.786,160.280
C07069=1014.598,357.022,346.067,171.099,51.789,160.279
C07070=1014.590,356.775,346.104,171.090,51.793,160.279
C07071=1014.583,356.527,346.142,171.081,51.796,160.278
C07072=1014.576,356.280,346.179,171.074,51.800,160.277
C07073=1014.568,356.033,346.216,171.065,51.803,160.276
C07074=1014.561,355.786,346.254,171.056,51.807,160.276
C07075=1014.554,355.539,346.291,171.049,51.811,160.275
C07076=1014.546,355.291,346.328,171.040,51.814,160.274
C07077=1014.538,355.045,346.365,171.031,51.819,160.274
C07078=1014.531,354.797,346.403,171.023,51.822,160.273
C07079=1014.524,354.550,346.440,171.014,51.826,160.272
C07080=1014.517,354.303,346.478,171.006,51.830,160.272
C07081=1014.509,354.056,346.514,170.998,51.833,160.271
C07082=1014.502,353.809,346.551,170.989,51.837,160.270
C07083=1014.494,353.520,346.594,170.980,51.841,160.270
C07084=1014.484,353.231,346.638,170.970,51.845,160.269
C07085=1014.477,352.943,346.681,170.961,51.850,160.268
C07086=1014.468,352.653,346.724,170.951,51.854,160.268
C07087=1014.460,352.406,346.761,170.943,51.858,160.267
C07088=1014.453,352.158,346.798,170.934,51.862,160.266
C07089=1014.446,351.912,346.834,170.926,51.866,160.266
C07090=1014.439,351.665,346.871,170.917,51.869,160.265
C07091=1014.431,351.417,346.908,170.909,51.873,160.264
C07092=1014.424,351.170,346.945,170.901,51.877,160.264
C07093=1014.417,350.923,346.981,170.893,51.881,160.263
C07094=1014.410,350.676,347.018,170.885,51.885,160.263
C07095=1014.402,350.429,347.055,170.877,51.889,160.262
C07096=1014.396,350.182,347.091,170.868,51.893,160.261
C07097=1014.388,349.934,347.127,170.861,51.897,160.261
C07098=1014.381,349.686,347.164,170.852,51.901,160.260
C07099=1014.374,349.440,347.201,170.845,51.905,160.260
C07100=1014.367,349.193,347.238,170.836,51.909,160.259
C07101=1014.359,348.945,347.274,170.828,51.913,160.258
C07102=1014.353,348.698,347.310,170.820,51.917,160.258
C07103=1014.345,348.451,347.347,170.812,51.921,160.257
C07104=1014.339,348.204,347.383,170.804,51.925,160.257
C07105=1014.331,347.956,347.419,170.796,51.929,160.256
C07106=1014.324,347.708,347.456,170.788,51.933,160.256
C07107=1014.317,347.462,347.492,170.780,51.937,160.255
C07108=1014.310,347.214,347.529,170.773,51.941,160.255
C07109=1014.303,346.967,347.565,170.764,51.945,160.254
C07110=1014.296,346.719,347.601,170.756,51.949,160.254
C07111=1014.289,346.473,347.637,170.748,51.953,160.253
C07112=1014.282,346.225,347.674,170.741,51.957,160.253
C07113=1014.275,345.978,347.710,170.732,51.961,160.252
C07114=1014.268,345.731,347.745,170.724,51.966,160.252
C07115=1014.261,345.483,347.781,170.716,51.970,160.251
C07116=1014.254,345.236,347.818,170.708,51.974,160.251
C07117=1014.247,344.989,347.854,170.701,51.978,160.250
C07118=1014.240,344.741,347.889,170.693,51.983,160.250
C07119=1014.233,344.494,347.926,170.685,51.986,160.249
C07120=1014.226,344.246,347.961,170.677,51.991,160.249
C07121=1014.219,344.000,347.997,170.670,51.995,160.248
C07122=1014.211,343.752,348.033,170.661,51.999,160.248
C07123=1014.205,343.504,348.069,170.654,52.004,160.247
C07124=1014.198,343.258,348.105,170.645,52.008,160.247
C07125=1014.191,343.010,348.140,170.638,52.012,160.246
C07126=1014.184,342.763,348.176,170.630,52.017,160.246
C07127=1014.178,342.515,348.212,170.623,52.021,160.246
C07128=1014.171,342.268,348.248,170.614,52.025,160.245
C07129=1014.163,342.020,348.283,170.607,52.029,160.245
C07130=1014.157,341.773,348.318,170.599,52.034,160.244
C07131=1014.150,341.526,348.354,170.592,52.038,160.244
C07132=1014.143,341.279,348.390,170.583,52.042,160.243
C07133=1014.136,341.031,348.425,170.576,52.047,160.243
C07134=1014.129,340.783,348.460,170.568,52.051,160.243
C07135=1014.122,340.536,348.496,170.561,52.056,160.242
C07136=1014.116,340.289,348.531,170.554,52.060,160.242
C07137=1014.109,340.041,348.567,170.546,52.065,160.241
C07138=1014.103,339.794,348.602,170.539,52.069,160.241
C07139=1014.095,339.546,348.638,170.530,52.073,160.240
C07140=1014.088,339.299,348.674,170.523,52.077,160.240
C07141=1014.081,339.052,348.709,170.515,52.082,160.240
C07142=1014.075,338.805,348.744,170.508,52.086,160.239
C07143=1014.067,338.513,348.785,170.499,52.092,160.239
C07144=1014.059,338.221,348.827,170.490,52.097,160.239
C07145=1014.052,337.930,348.868,170.481,52.103,160.238
C07146=1014.044,337.638,348.910,170.472,52.108,160.238
C07147=1014.036,337.391,348.944,170.465,52.112,160.237
C07148=1014.029,337.143,348.979,170.457,52.117,160.237
C07149=1014.022,336.896,349.014,170.450,52.122,160.237
C07150=1014.016,336.648,349.049,170.442,52.127,160.236
C07151=1014.009,336.401,349.084,170.435,52.131,160.236
C07152=1014.002,336.153,349.119,170.426,52.136,160.236
C07153=1013.996,335.906,349.154,170.420,52.141,160.236
C07154=1013.989,335.658,349.189,170.412,52.146,160.235
C07155=1013.983,335.410,349.224,170.405,52.150,160.235
C07156=1013.976,335.163,349.259,170.397,52.154,160.234
C07157=1013.969,334.915,349.293,170.390,52.160,160.234
C07158=1013.963,334.668,349.328,170.383,52.164,160.234
C07159=1013.956,334.421,349.363,170.374,52.169,160.233
C07160=1013.949,334.173,349.397,170.368,52.174,160.233
C07161=1013.942,333.926,349.432,170.361,52.178,160.233
C07162=1013.936,333.678,349.467,170.353,52.183,160.233
C07163=1013.929,333.431,349.502,170.346,52.188,160.232
C07164=1013.923,333.183,349.536,170.338,52.192,160.232
C07165=1013.917,332.936,349.571,170.331,52.197,160.232
C07166=1013.910,332.688,349.605,170.324,52.202,160.232
C07167=1013.903,332.441,349.641,170.316,52.207,160.231
C07168=1013.897,332.193,349.675,170.309,52.211,160.231
C07169=1013.891,331.945,349.709,170.301,52.217,160.231
C07170=1013.883,331.698,349.744,170.294,52.221,160.230
C07171=1013.877,331.450,349.778,170.287,52.226,160.230
C07172=1013.871,331.203,349.812,170.280,52.231,160.230
C07173=1013.864,330.955,349.846,170.272,52.236,160.230
C07174=1013.857,330.707,349.880,170.265,52.241,160.230
C07175=1013.851,330.460,349.915,170.258,52.246,160.229
C07176=1013.844,330.213,349.949,170.251,52.251,160.229
C07177=1013.838,329.965,349.983,170.243,52.256,160.229
C07178=1013.831,329.717,350.018,170.236,52.261,160.229
C07179=1013.825,329.470,350.051,170.229,52.266,160.229
C07180=1013.818,329.222,350.086,170.222,52.271,160.228
C07181=1013.812,328.975,350.119,170.215,52.276,160.228
C07182=1013.805,328.727,350.153,170.207,52.281,160.228
C07183=1013.799,328.479,350.188,170.201,52.286,160.228
C07184=1013.792,328.232,350.221,170.194,52.291,160.228
C07185=1013.786,327.984,350.256,170.186,52.296,160.227
C07186=1013.780,327.737,350.290,170.179,52.301,160.227
C07187=1013.772,327.489,350.324,170.171,52.306,160.227
C07188=1013.767,327.242,350.358,170.165,52.311,160.227
C07189=1013.760,326.994,350.392,170.158,52.316,160.227
C07190=1013.754,326.746,350.425,170.150,52.322,160.226
C07191=1013.747,326.498,350.459,170.143,52.327,160.226
C07192=1013.742,326.251,350.493,170.137,52.332,160.226
C07193=1013.734,326.003,350.527,170.129,52.337,160.226
C07194=1013.728,325.756,350.561,170.122,52.342,160.226
C07195=1013.722,325.508,350.594,170.116,52.347,160.226
C07196=1013.715,325.261,350.628,170.108,52.352,160.225
C07197=1013.709,325.013,350.661,170.101,52.357,160.225
C07198=1013.702,324.765,350.695,170.093,52.363,160.225
C07199=1013.696,324.518,350.728,170.087,52.368,160.225
C07200=1013.689,324.270,350.761,170.080,52.374,160.225
C07201=1013.682,324.022,350.794,170.073,52.379,160.225
C07202=1013.676,323.775,350.829,170.066,52.384,160.225
C07203=1013.669,323.479,350.868,170.058,52.390,160.224
C07204=1013.660,323.183,350.907,170.050,52.397,160.224
C07205=1013.653,322.887,350.947,170.040,52.404,160.224
C07206=1013.645,322.591,350.987,170.032,52.410,160.224
C07207=1013.638,322.344,351.020,170.025,52.415,160.224
C07208=1013.632,322.096,351.053,170.019,52.421,160.224
C07209=1013.626,321.848,351.087,170.011,52.426,160.224
C07210=1013.620,321.600,351.120,170.005,52.431,160.224
C07211=1013.613,321.353,351.153,169.998,52.437,160.224
C07212=1013.606,321.105,351.186,169.991,52.442,160.224
C07213=1013.600,320.857,351.219,169.984,52.448,160.224
C07214=1013.594,320.609,351.252,169.977,52.453,160.223
C07215=1013.588,320.362,351.285,169.970,52.458,160.223
C07216=1013.581,320.113,351.318,169.964,52.464,160.223
C07217=1013.575,319.866,351.351,169.956,52.469,160.223
C07218=1013.568,319.619,351.384,169.950,52.475,160.223
C07219=1013.563,319.371,351.418,169.943,52.480,160.223
C07220=1013.556,319.123,351.450,169.936,52.486,160.223
C07221=1013.550,318.876,351.483,169.929,52.491,160.223
C07222=1013.544,318.628,351.516,169.922,52.497,160.223
C07223=1013.537,318.380,351.549,169.916,52.503,160.223
C07224=1013.531,318.132,351.582,169.909,52.508,160.223
C07225=1013.525,317.884,351.615,169.902,52.514,160.223
C07226=1013.519,317.637,351.648,169.895,52.519,160.223
C07227=1013.513,317.389,351.680,169.889,52.525,160.223
C07228=1013.506,317.142,351.713,169.881,52.531,160.223
C07229=1013.500,316.894,351.746,169.875,52.536,160.223
C07230=1013.494,316.646,351.779,169.869,52.542,160.223
C07231=1013.488,316.398,351.811,169.861,52.548,160.223
C07232=1013.482,316.150,351.844,169.855,52.553,160.223
C07233=1013.476,315.903,351.877,169.848,52.558,160.223
C07234=1013.470,315.655,351.910,169.841,52.564,160.223
C07235=1013.464,315.407,351.943,169.835,52.570,160.223
C07236=1013.458,315.159,351.975,169.829,52.576,160.223
C07237=1013.452,314.911,352.008,169.821,52.581,160.223
C07238=1013.445,314.664,352.040,169.815,52.587,160.223
C07239=1013.439,314.416,352.073,169.808,52.593,160.223
C07240=1013.433,314.168,352.105,169.801,52.599,160.223
C07241=1013.428,313.920,352.139,169.795,52.605,160.223
C07242=1013.422,313.673,352.171,169.788,52.610,160.223
C07243=1013.416,313.425,352.203,169.781,52.616,160.223
C07244=1013.410,313.177,352.236,169.775,52.621,160.223
C07245=1013.403,312.930,352.268,169.768,52.627,160.223
C07246=1013.397,312.682,352.300,169.761,52.633,160.223
C07247=1013.392,312.434,352.334,169.755,52.639,160.223
C07248=1013.386,312.186,352.365,169.749,52.645,160.223
C07249=1013.380,311.939,352.398,169.741,52.651,160.223
C07250=1013.374,311.691,352.431,169.735,52.656,160.223
C07251=1013.368,311.443,352.463,169.729,52.662,160.223
C07252=1013.363,311.196,352.496,169.723,52.668,160.223
C07253=1013.357,310.947,352.528,169.715,52.674,160.223
C07254=1013.351,310.700,352.561,169.709,52.680,160.223
C07255=1013.345,310.452,352.593,169.703,52.685,160.223
C07256=1013.339,310.204,352.624,169.696,52.691,160.223
C07257=1013.333,309.956,352.657,169.689,52.697,160.223
C07258=1013.328,309.708,352.690,169.683,52.703,160.223
C07259=1013.322,309.461,352.722,169.676,52.709,160.223
C07260=1013.316,309.213,352.754,169.670,52.715,160.224
C07261=1013.310,308.965,352.786,169.664,52.721,160.224
C07262=1013.304,308.717,352.817,169.657,52.727,160.224
C07263=1013.297,308.427,352.855,169.650,52.734,160.224
